METHOD lockstep_move_max
VAR_INPUT
	LockstepGroup	: USINT := 1; // The address of the lockstep group must be in the range 1 to lockstep.numgroups; lockstep.numgroups: the number of lockstep groupss; Valid Values: 0 to 2
	max_speed 		: UDINT := ZaberConfiguration.MaxDynamics.Velocity;
	accel			: UDINT	:= ZaberConfiguration.MaxDynamics.Accel;
END_VAR
IF ZaberStatus.ComponentStatus.iLastCommand <> 0 THEN
	ZaberStatus.ComponentStatus.iLastCommand.P_CommandStatus.LastCommandMessage := Base.F_GetLastWordInString(__POUNAME());
END_IF

IF NOT _DispatchValid() THEN
	RETURN;
ELSE
	_ClearTempString();
	ZaberCommand.stringval := Tc2_Standard.CONCAT(STR1 := ZaberConfiguration.sControllerRef, STR2 := ' ');
	ZaberCommand.stringval := Tc2_Standard.CONCAT(STR1 := ZaberCommand.stringval, STR2 := Base.F_GetFirstWordInString(sInput := SUPER^._iCommandConfiguration[ZaberStatus.ZaberMethodDispatch].P_CommandConfiguration.CommandDescription));
	ZaberCommand.stringval := Tc2_Standard.CONCAT(STR1 := ZaberCommand.stringval, STR2 := ' ');
	ZaberCommand.stringval := Tc2_Standard.CONCAT(STR1 := ZaberCommand.stringval, STR2 := USINT_TO_STRING(LockstepGroup));
	ZaberCommand.stringval := Tc2_Standard.CONCAT(STR1 := ZaberCommand.stringval, STR2 := ' ');
	ZaberCommand.stringval := Tc2_Standard.CONCAT(STR1 := ZaberCommand.stringval, STR2 := F_GetAllButFirstWord(sInput := SUPER^._iCommandConfiguration[ZaberStatus.ZaberMethodDispatch].P_CommandConfiguration.CommandDescription));
	ZaberCommand.stringval := Tc2_Standard.CONCAT(STR1 := ZaberCommand.stringval, STR2 := ' ');
	ZaberCommand.stringval := Tc2_Standard.CONCAT(STR1 := ZaberCommand.stringval, STR2 := UDINT_TO_STRING(max_speed));
	ZaberCommand.stringval := Tc2_Standard.CONCAT(STR1 := ZaberCommand.stringval, STR2 := ' ');
	ZaberCommand.stringval := Tc2_Standard.CONCAT(STR1 := ZaberCommand.stringval, STR2 := UDINT_TO_STRING(accel));
	
	IF iBufferSend <> 0 AND __QUERYINTERFACE(iBufferSend, testIBufferSend) THEN
		iBufferSend.AddObject(RefObject := ZaberCommand);
	END_IF
END_IF
END_METHOD

METHOD lockstep_move_min
VAR_INPUT
	LockstepGroup	: USINT := 1; // The address of the lockstep group must be in the range 1 to lockstep.numgroups; lockstep.numgroups: the number of lockstep groupss; Valid Values: 0 to 2
	max_speed 		: UDINT := ZaberConfiguration.MaxDynamics.Velocity;
	accel			: UDINT := ZaberConfiguration.MaxDynamics.Accel;
END_VAR
IF ZaberStatus.ComponentStatus.iLastCommand <> 0 THEN
	ZaberStatus.ComponentStatus.iLastCommand.P_CommandStatus.LastCommandMessage := Base.F_GetLastWordInString(__POUNAME());
END_IF

IF NOT _DispatchValid() THEN
	RETURN;
ELSE
	_ClearTempString();
	ZaberCommand.stringval := Tc2_Standard.CONCAT(STR1 := ZaberConfiguration.sControllerRef, STR2 := ' ');
	ZaberCommand.stringval := Tc2_Standard.CONCAT(STR1 := ZaberCommand.stringval, STR2 := Base.F_GetFirstWordInString(sInput := SUPER^._iCommandConfiguration[ZaberStatus.ZaberMethodDispatch].P_CommandConfiguration.CommandDescription));
	ZaberCommand.stringval := Tc2_Standard.CONCAT(STR1 := ZaberCommand.stringval, STR2 := ' ');
	ZaberCommand.stringval := Tc2_Standard.CONCAT(STR1 := ZaberCommand.stringval, STR2 := USINT_TO_STRING(LockstepGroup));
	ZaberCommand.stringval := Tc2_Standard.CONCAT(STR1 := ZaberCommand.stringval, STR2 := ' ');
	ZaberCommand.stringval := Tc2_Standard.CONCAT(STR1 := ZaberCommand.stringval, STR2 := F_GetAllButFirstWord(sInput := SUPER^._iCommandConfiguration[ZaberStatus.ZaberMethodDispatch].P_CommandConfiguration.CommandDescription));
	ZaberCommand.stringval := Tc2_Standard.CONCAT(STR1 := ZaberCommand.stringval, STR2 := ' ');
	ZaberCommand.stringval := Tc2_Standard.CONCAT(STR1 := ZaberCommand.stringval, STR2 := UDINT_TO_STRING(max_speed));
	ZaberCommand.stringval := Tc2_Standard.CONCAT(STR1 := ZaberCommand.stringval, STR2 := ' ');
	ZaberCommand.stringval := Tc2_Standard.CONCAT(STR1 := ZaberCommand.stringval, STR2 := UDINT_TO_STRING(accel));
	
	IF iBufferSend <> 0 AND __QUERYINTERFACE(iBufferSend, testIBufferSend) THEN
		iBufferSend.AddObject(RefObject := ZaberCommand);
	END_IF
END_IF
END_METHOD

METHOD lockstep_move_sin
VAR_INPUT
	LockstepGroup	: USINT := 1; // The address of the lockstep group must be in the range 1 to lockstep.numgroups; lockstep.numgroups: the number of lockstep groupss; Valid Values: 0 to 2
	amplitude		: LREAL := ZaberConfiguration.SinParameters.Amplitude; // Amplitude of the sinusoidal motion
	period	 		: LREAL := ZaberConfiguration.SinParameters.Period; // Period of the sinusoidal motion in milliseconds and to one decimal place; Must be in the range 0.2 to 429,496,729.5
	count			: LREAL := ZaberConfiguration.SinParameters.Count; // Number of repeated cycles (optional); Must be a multiple of 0.5 in the range 0.5 to 2,147,483,647 (versions 7.29 and above)
END_VAR
IF ZaberStatus.ComponentStatus.iLastCommand <> 0 THEN
	ZaberStatus.ComponentStatus.iLastCommand.P_CommandStatus.LastCommandMessage := Base.F_GetLastWordInString(__POUNAME());
END_IF

IF NOT _DispatchValid() THEN
	RETURN;
ELSE
	_ClearTempString();
	ZaberCommand.stringval := Tc2_Standard.CONCAT(STR1 := ZaberConfiguration.sControllerRef, STR2 := ' ');
	ZaberCommand.stringval := Tc2_Standard.CONCAT(STR1 := ZaberCommand.stringval, STR2 := Base.F_GetFirstWordInString(sInput := SUPER^._iCommandConfiguration[ZaberStatus.ZaberMethodDispatch].P_CommandConfiguration.CommandDescription));
	ZaberCommand.stringval := Tc2_Standard.CONCAT(STR1 := ZaberCommand.stringval, STR2 := ' ');
	ZaberCommand.stringval := Tc2_Standard.CONCAT(STR1 := ZaberCommand.stringval, STR2 := USINT_TO_STRING(LockstepGroup));
	ZaberCommand.stringval := Tc2_Standard.CONCAT(STR1 := ZaberCommand.stringval, STR2 := ' ');
	ZaberCommand.stringval := Tc2_Standard.CONCAT(STR1 := ZaberCommand.stringval, STR2 := F_GetAllButFirstWord(sInput := SUPER^._iCommandConfiguration[ZaberStatus.ZaberMethodDispatch].P_CommandConfiguration.CommandDescription));
	ZaberCommand.stringval := Tc2_Standard.CONCAT(STR1 := ZaberCommand.stringval, STR2 := ' ');
	ZaberCommand.stringval := Tc2_Standard.CONCAT(STR1 := ZaberCommand.stringval, STR2 := LREAL_TO_STRING(amplitude));
	ZaberCommand.stringval := Tc2_Standard.CONCAT(STR1 := ZaberCommand.stringval, STR2 := ' ');
	ZaberCommand.stringval := Tc2_Standard.CONCAT(STR1 := ZaberCommand.stringval, STR2 := LREAL_TO_STRING(period));
	ZaberCommand.stringval := Tc2_Standard.CONCAT(STR1 := ZaberCommand.stringval, STR2 := ' ');
	ZaberCommand.stringval := Tc2_Standard.CONCAT(STR1 := ZaberCommand.stringval, STR2 := LREAL_TO_STRING(count));
	
	IF iBufferSend <> 0 AND __QUERYINTERFACE(iBufferSend, testIBufferSend) THEN
		iBufferSend.AddObject(RefObject := ZaberCommand);
	END_IF
END_IF
END_METHOD

METHOD move_abs
VAR_INPUT
	position	: UDINT := ZaberConfiguration.SetDynamics.Position;
	max_speed 	: UDINT := ZaberConfiguration.MaxDynamics.Velocity;
	accel		: UDINT := ZaberConfiguration.MaxDynamics.Accel;
END_VAR
IF ZaberStatus.ComponentStatus.iLastCommand <> 0 THEN
	ZaberStatus.ComponentStatus.iLastCommand.P_CommandStatus.LastCommandMessage := Base.F_GetLastWordInString(__POUNAME());
END_IF

IF NOT _DispatchValid() THEN
	RETURN;
ELSE
	_BuildCommandStringNoArgs();
	ZaberCommand.stringval := Tc2_Standard.CONCAT(STR1 := ZaberCommand.stringval, STR2 := ' ');
	ZaberCommand.stringval := Tc2_Standard.CONCAT(STR1 := ZaberCommand.stringval, STR2 := UDINT_TO_STRING(position));
	ZaberCommand.stringval := Tc2_Standard.CONCAT(STR1 := ZaberCommand.stringval, STR2 := ' ');
	ZaberCommand.stringval := Tc2_Standard.CONCAT(STR1 := ZaberCommand.stringval, STR2 := UDINT_TO_STRING(max_speed));
	ZaberCommand.stringval := Tc2_Standard.CONCAT(STR1 := ZaberCommand.stringval, STR2 := ' ');
	ZaberCommand.stringval := Tc2_Standard.CONCAT(STR1 := ZaberCommand.stringval, STR2 := UDINT_TO_STRING(accel));

	IF iBufferSend <> 0 AND __QUERYINTERFACE(iBufferSend, testIBufferSend) THEN
		iBufferSend.AddObject(RefObject := ZaberCommand);
	END_IF
END_IF
END_METHOD

METHOD move_index_next
IF ZaberStatus.ComponentStatus.iLastCommand <> 0 THEN
	ZaberStatus.ComponentStatus.iLastCommand.P_CommandStatus.LastCommandMessage := Base.F_GetLastWordInString(__POUNAME());
END_IF

IF NOT _DispatchValid() THEN
	RETURN;
ELSE
	_BuildCommandStringNoArgs();
	
	IF iBufferSend <> 0 AND __QUERYINTERFACE(iBufferSend, testIBufferSend) THEN
		iBufferSend.AddObject(RefObject := ZaberCommand);
	END_IF
END_IF
END_METHOD

METHOD move_index_prev
IF ZaberStatus.ComponentStatus.iLastCommand <> 0 THEN
	ZaberStatus.ComponentStatus.iLastCommand.P_CommandStatus.LastCommandMessage := Base.F_GetLastWordInString(__POUNAME());
END_IF

IF NOT _DispatchValid() THEN
	RETURN;
ELSE
	_BuildCommandStringNoArgs();
	
	IF iBufferSend <> 0 AND __QUERYINTERFACE(iBufferSend, testIBufferSend) THEN
		iBufferSend.AddObject(RefObject := ZaberCommand);
	END_IF
END_IF
END_METHOD

METHOD move_max
IF ZaberStatus.ComponentStatus.iLastCommand <> 0 THEN
	ZaberStatus.ComponentStatus.iLastCommand.P_CommandStatus.LastCommandMessage := Base.F_GetLastWordInString(__POUNAME());
END_IF

IF NOT _DispatchValid() THEN
	RETURN;
ELSE
	_BuildCommandStringNoArgs();
	
	IF iBufferSend <> 0 AND __QUERYINTERFACE(iBufferSend, testIBufferSend) THEN
		iBufferSend.AddObject(RefObject := ZaberCommand);
	END_IF
END_IF
END_METHOD

METHOD move_min
IF ZaberStatus.ComponentStatus.iLastCommand <> 0 THEN
	ZaberStatus.ComponentStatus.iLastCommand.P_CommandStatus.LastCommandMessage := Base.F_GetLastWordInString(__POUNAME());
END_IF

IF NOT _DispatchValid() THEN
	RETURN;
ELSE
	_BuildCommandStringNoArgs();
	
	IF iBufferSend <> 0 AND __QUERYINTERFACE(iBufferSend, testIBufferSend) THEN
		iBufferSend.AddObject(RefObject := ZaberCommand);
	END_IF
END_IF
END_METHOD

METHOD move_scan_track_once
IF ZaberStatus.ComponentStatus.iLastCommand <> 0 THEN
	ZaberStatus.ComponentStatus.iLastCommand.P_CommandStatus.LastCommandMessage := Base.F_GetLastWordInString(__POUNAME());
END_IF

IF NOT _DispatchValid() THEN
	RETURN;
ELSE
	_BuildCommandStringNoArgs();
	
	IF iBufferSend <> 0 AND __QUERYINTERFACE(iBufferSend, testIBufferSend) THEN
		iBufferSend.AddObject(RefObject := ZaberCommand);
	END_IF
END_IF
END_METHOD

METHOD move_sin
VAR_INPUT
	amplitude		: LREAL; // Amplitude of the sinusoidal motion
	period	 		: LREAL; // Period of the sinusoidal motion in milliseconds and to one decimal place; Must be in the range 0.2 to 429,496,729.5
	count			: LREAL; // Number of repeated cycles (optional); Must be a multiple of 0.5 in the range 0.5 to 2,147,483,647 (versions 7.29 and above)
END_VAR
IF ZaberStatus.ComponentStatus.iLastCommand <> 0 THEN
	ZaberStatus.ComponentStatus.iLastCommand.P_CommandStatus.LastCommandMessage := Base.F_GetLastWordInString(__POUNAME());
END_IF

IF NOT _DispatchValid() THEN
	RETURN;
ELSE
	_ClearTempString();
	ZaberCommand.stringval := Tc2_Standard.CONCAT(STR1 := ZaberConfiguration.sControllerRef, STR2 := ' ');
	ZaberCommand.stringval := Tc2_Standard.CONCAT(STR1 := ZaberCommand.stringval, STR2 := UINT_TO_STRING(ZaberConfiguration.AxisRef));
	ZaberCommand.stringval := Tc2_Standard.CONCAT(STR1 := ZaberCommand.stringval, STR2 := ' ');
	ZaberCommand.stringval := Tc2_Standard.CONCAT(STR1 := ZaberCommand.stringval, STR2 := SUPER^._iCommandConfiguration[ZaberStatus.ZaberMethodDispatch].P_CommandConfiguration.CommandDescription);
	ZaberCommand.stringval := Tc2_Standard.CONCAT(STR1 := ZaberCommand.stringval, STR2 := ' ');
	ZaberCommand.stringval := Tc2_Standard.CONCAT(STR1 := ZaberCommand.stringval, STR2 := LREAL_TO_STRING(amplitude));
	ZaberCommand.stringval := Tc2_Standard.CONCAT(STR1 := ZaberCommand.stringval, STR2 := ' ');
	ZaberCommand.stringval := Tc2_Standard.CONCAT(STR1 := ZaberCommand.stringval, STR2 := LREAL_TO_STRING(period));
	ZaberCommand.stringval := Tc2_Standard.CONCAT(STR1 := ZaberCommand.stringval, STR2 := ' ');
	ZaberCommand.stringval := Tc2_Standard.CONCAT(STR1 := ZaberCommand.stringval, STR2 := LREAL_TO_STRING(count));
	
	IF iBufferSend <> 0 AND __QUERYINTERFACE(iBufferSend, testIBufferSend) THEN
		iBufferSend.AddObject(RefObject := ZaberCommand);
	END_IF
END_IF
END_METHOD

METHOD move_track
IF ZaberStatus.ComponentStatus.iLastCommand <> 0 THEN
	ZaberStatus.ComponentStatus.iLastCommand.P_CommandStatus.LastCommandMessage := Base.F_GetLastWordInString(__POUNAME());
END_IF

IF NOT _DispatchValid() THEN
	RETURN;
ELSE
	_BuildCommandStringNoArgs();
	
	IF iBufferSend <> 0 AND __QUERYINTERFACE(iBufferSend, testIBufferSend) THEN
		iBufferSend.AddObject(RefObject := ZaberCommand);
	END_IF
END_IF
END_METHOD

METHOD move_vel
VAR_INPUT
	velocity		: DINT;
	accel			: UDINT;
END_VAR
IF ZaberStatus.ComponentStatus.iLastCommand <> 0 THEN
	ZaberStatus.ComponentStatus.iLastCommand.P_CommandStatus.LastCommandMessage := Base.F_GetLastWordInString(__POUNAME());
END_IF

IF NOT _DispatchValid() THEN
	RETURN;
ELSE
	_ClearTempString();
	ZaberCommand.stringval := Tc2_Standard.CONCAT(STR1 := ZaberConfiguration.sControllerRef, STR2 := ' ');
	ZaberCommand.stringval := Tc2_Standard.CONCAT(STR1 := ZaberCommand.stringval, STR2 := UINT_TO_STRING(ZaberConfiguration.AxisRef));
	ZaberCommand.stringval := Tc2_Standard.CONCAT(STR1 := ZaberCommand.stringval, STR2 := ' ');
	ZaberCommand.stringval := Tc2_Standard.CONCAT(STR1 := ZaberCommand.stringval, STR2 := SUPER^._iCommandConfiguration[ZaberStatus.ZaberMethodDispatch].P_CommandConfiguration.CommandDescription);
	ZaberCommand.stringval := Tc2_Standard.CONCAT(STR1 := ZaberCommand.stringval, STR2 := ' ');
	ZaberCommand.stringval := Tc2_Standard.CONCAT(STR1 := ZaberCommand.stringval, STR2 := DINT_TO_STRING(velocity));
	ZaberCommand.stringval := Tc2_Standard.CONCAT(STR1 := ZaberCommand.stringval, STR2 := ' ');
	ZaberCommand.stringval := Tc2_Standard.CONCAT(STR1 := ZaberCommand.stringval, STR2 := UDINT_TO_STRING(accel));
	
	IF iBufferSend <> 0 AND __QUERYINTERFACE(iBufferSend, testIBufferSend) THEN
		iBufferSend.AddObject(RefObject := ZaberCommand);
	END_IF
END_IF
END_METHOD

METHOD pvt_buffer_list
IF ZaberStatus.ComponentStatus.iLastCommand <> 0 THEN
	ZaberStatus.ComponentStatus.iLastCommand.P_CommandStatus.LastCommandMessage := Base.F_GetLastWordInString(__POUNAME());
END_IF

IF NOT _DispatchValid() THEN
	RETURN;
ELSE
	_BuildCommandStringNoArgs();
	
	IF iBufferSend <> 0 AND __QUERYINTERFACE(iBufferSend, testIBufferSend) THEN
		iBufferSend.AddObject(RefObject := ZaberCommand);
	END_IF
END_IF
END_METHOD

METHOD renumber
IF ZaberStatus.ComponentStatus.iLastCommand <> 0 THEN
	ZaberStatus.ComponentStatus.iLastCommand.P_CommandStatus.LastCommandMessage := Base.F_GetLastWordInString(__POUNAME());
END_IF

IF NOT _DispatchValid() THEN
	RETURN;
ELSE
	_BuildCommandStringNoArgs();
	
	IF iBufferSend <> 0 AND __QUERYINTERFACE(iBufferSend, testIBufferSend) THEN
		iBufferSend.AddObject(RefObject := ZaberCommand);
	END_IF
END_IF
END_METHOD

METHOD scope_clear
IF ZaberStatus.ComponentStatus.iLastCommand <> 0 THEN
	ZaberStatus.ComponentStatus.iLastCommand.P_CommandStatus.LastCommandMessage := Base.F_GetLastWordInString(__POUNAME());
END_IF

IF NOT _DispatchValid() THEN
	RETURN;
ELSE
	_BuildCommandStringNoArgs();
	
	IF iBufferSend <> 0 AND __QUERYINTERFACE(iBufferSend, testIBufferSend) THEN
		iBufferSend.AddObject(RefObject := ZaberCommand);
	END_IF
END_IF
END_METHOD

METHOD scope_print
IF ZaberStatus.ComponentStatus.iLastCommand <> 0 THEN
	ZaberStatus.ComponentStatus.iLastCommand.P_CommandStatus.LastCommandMessage := Base.F_GetLastWordInString(__POUNAME());
END_IF

IF NOT _DispatchValid() THEN
	RETURN;
ELSE
	_BuildCommandStringNoArgs();
	
	IF iBufferSend <> 0 AND __QUERYINTERFACE(iBufferSend, testIBufferSend) THEN
		iBufferSend.AddObject(RefObject := ZaberCommand);
	END_IF
END_IF
END_METHOD

METHOD scope_stop
IF ZaberStatus.ComponentStatus.iLastCommand <> 0 THEN
	ZaberStatus.ComponentStatus.iLastCommand.P_CommandStatus.LastCommandMessage := Base.F_GetLastWordInString(__POUNAME());
END_IF

IF NOT _DispatchValid() THEN
	RETURN;
ELSE
	_BuildCommandStringNoArgs();
	
	IF iBufferSend <> 0 AND __QUERYINTERFACE(iBufferSend, testIBufferSend) THEN
		iBufferSend.AddObject(RefObject := ZaberCommand);
	END_IF
END_IF
END_METHOD

METHOD set_comm_checksum
VAR_INPUT
	Value	: INT := 1; //0 = Disabled, 1 = Enabled, 2 = Automatic
END_VAR
IF ZaberStatus.ComponentStatus.iLastCommand <> 0 THEN
	ZaberStatus.ComponentStatus.iLastCommand.P_CommandStatus.LastCommandMessage := Base.F_GetLastWordInString(__POUNAME());
END_IF

IF NOT _DispatchValid() THEN
	RETURN;
ELSE
	_BuildCommandStringNoArgs();
	ZaberCommand.stringval := Tc2_Standard.CONCAT(STR1 := ZaberCommand.stringval, STR2 := ' ');
	ZaberCommand.stringval := Tc2_Standard.CONCAT(STR1 := ZaberCommand.stringval, STR2 := INT_TO_STRING(Value));
	
	IF iBufferSend <> 0 AND __QUERYINTERFACE(iBufferSend, testIBufferSend) THEN
		iBufferSend.AddObject(RefObject := ZaberCommand);
	END_IF
END_IF
END_METHOD

METHOD stop
IF ZaberStatus.ComponentStatus.iLastCommand <> 0 THEN
	ZaberStatus.ComponentStatus.iLastCommand.P_CommandStatus.LastCommandMessage := Base.F_GetLastWordInString(__POUNAME());
END_IF

IF NOT _DispatchValid() THEN
	RETURN;
ELSE
	_BuildCommandStringNoArgs();
	
	IF iBufferSend <> 0 AND __QUERYINTERFACE(iBufferSend, testIBufferSend) THEN
		iBufferSend.AddObject(RefObject := ZaberCommand);
	END_IF
END_IF
END_METHOD

METHOD storage_erase
IF ZaberStatus.ComponentStatus.iLastCommand <> 0 THEN
	ZaberStatus.ComponentStatus.iLastCommand.P_CommandStatus.LastCommandMessage := Base.F_GetLastWordInString(__POUNAME());
END_IF

IF NOT _DispatchValid() THEN
	RETURN;
ELSE
	_BuildCommandStringNoArgs();
	
	IF iBufferSend <> 0 AND __QUERYINTERFACE(iBufferSend, testIBufferSend) THEN
		iBufferSend.AddObject(RefObject := ZaberCommand);
	END_IF
END_IF
END_METHOD

METHOD storage_print
IF ZaberStatus.ComponentStatus.iLastCommand <> 0 THEN
	ZaberStatus.ComponentStatus.iLastCommand.P_CommandStatus.LastCommandMessage := Base.F_GetLastWordInString(__POUNAME());
END_IF

IF NOT _DispatchValid() THEN
	RETURN;
ELSE
	_BuildCommandStringNoArgs();
	
	IF iBufferSend <> 0 AND __QUERYINTERFACE(iBufferSend, testIBufferSend) THEN
		iBufferSend.AddObject(RefObject := ZaberCommand);
	END_IF
END_IF
END_METHOD

METHOD stream_buffer_list
IF ZaberStatus.ComponentStatus.iLastCommand <> 0 THEN
	ZaberStatus.ComponentStatus.iLastCommand.P_CommandStatus.LastCommandMessage := Base.F_GetLastWordInString(__POUNAME());
END_IF

IF NOT _DispatchValid() THEN
	RETURN;
ELSE
	_BuildCommandStringNoArgs();
	
	IF iBufferSend <> 0 AND __QUERYINTERFACE(iBufferSend, testIBufferSend) THEN
		iBufferSend.AddObject(RefObject := ZaberCommand);
	END_IF
END_IF
END_METHOD

METHOD system_errors
IF ZaberStatus.ComponentStatus.iLastCommand <> 0 THEN
	ZaberStatus.ComponentStatus.iLastCommand.P_CommandStatus.LastCommandMessage := Base.F_GetLastWordInString(__POUNAME());
END_IF

IF NOT _DispatchValid() THEN
	RETURN;
ELSE
	_BuildCommandStringNoArgs();
	
	IF iBufferSend <> 0 AND __QUERYINTERFACE(iBufferSend, testIBufferSend) THEN
		iBufferSend.AddObject(RefObject := ZaberCommand);
	END_IF
END_IF
END_METHOD

METHOD system_factoryreset
IF ZaberStatus.ComponentStatus.iLastCommand <> 0 THEN
	ZaberStatus.ComponentStatus.iLastCommand.P_CommandStatus.LastCommandMessage := Base.F_GetLastWordInString(__POUNAME());
END_IF

IF NOT _DispatchValid() THEN
	RETURN;
ELSE
	_BuildCommandStringNoArgs();
	
	IF iBufferSend <> 0 AND __QUERYINTERFACE(iBufferSend, testIBufferSend) THEN
		iBufferSend.AddObject(RefObject := ZaberCommand);
	END_IF
END_IF
END_METHOD

METHOD system_reset
IF ZaberStatus.ComponentStatus.iLastCommand <> 0 THEN
	ZaberStatus.ComponentStatus.iLastCommand.P_CommandStatus.LastCommandMessage := Base.F_GetLastWordInString(__POUNAME());
END_IF

IF NOT _DispatchValid() THEN
	RETURN;
ELSE
	_BuildCommandStringNoArgs();
	
	IF iBufferSend <> 0 AND __QUERYINTERFACE(iBufferSend, testIBufferSend) THEN
		iBufferSend.AddObject(RefObject := ZaberCommand);
	END_IF
END_IF
END_METHOD

METHOD system_restore
IF ZaberStatus.ComponentStatus.iLastCommand <> 0 THEN
	ZaberStatus.ComponentStatus.iLastCommand.P_CommandStatus.LastCommandMessage := Base.F_GetLastWordInString(__POUNAME());
END_IF

IF NOT _DispatchValid() THEN
	RETURN;
ELSE
	_BuildCommandStringNoArgs();
	
	IF iBufferSend <> 0 AND __QUERYINTERFACE(iBufferSend, testIBufferSend) THEN
		iBufferSend.AddObject(RefObject := ZaberCommand);
	END_IF
END_IF
END_METHOD

METHOD tools_echo
IF ZaberStatus.ComponentStatus.iLastCommand <> 0 THEN
	ZaberStatus.ComponentStatus.iLastCommand.P_CommandStatus.LastCommandMessage := Base.F_GetLastWordInString(__POUNAME());
END_IF

IF NOT _DispatchValid() THEN
	RETURN;
ELSE
	_BuildCommandStringNoArgs();
	
	IF iBufferSend <> 0 AND __QUERYINTERFACE(iBufferSend, testIBufferSend) THEN
		iBufferSend.AddObject(RefObject := ZaberCommand);
	END_IF
END_IF
END_METHOD

METHOD tools_findrange
IF ZaberStatus.ComponentStatus.iLastCommand <> 0 THEN
	ZaberStatus.ComponentStatus.iLastCommand.P_CommandStatus.LastCommandMessage := Base.F_GetLastWordInString(__POUNAME());
END_IF

IF NOT _DispatchValid() THEN
	RETURN;
ELSE
	_BuildCommandStringNoArgs();
	
	IF iBufferSend <> 0 AND __QUERYINTERFACE(iBufferSend, testIBufferSend) THEN
		iBufferSend.AddObject(RefObject := ZaberCommand);
	END_IF
END_IF
END_METHOD

METHOD tools_gotolimit
IF ZaberStatus.ComponentStatus.iLastCommand <> 0 THEN
	ZaberStatus.ComponentStatus.iLastCommand.P_CommandStatus.LastCommandMessage := Base.F_GetLastWordInString(__POUNAME());
END_IF

IF NOT _DispatchValid() THEN
	RETURN;
ELSE
	_BuildCommandStringNoArgs();
	
	IF iBufferSend <> 0 AND __QUERYINTERFACE(iBufferSend, testIBufferSend) THEN
		iBufferSend.AddObject(RefObject := ZaberCommand);
	END_IF
END_IF
END_METHOD

METHOD tools_parking
IF ZaberStatus.ComponentStatus.iLastCommand <> 0 THEN
	ZaberStatus.ComponentStatus.iLastCommand.P_CommandStatus.LastCommandMessage := Base.F_GetLastWordInString(__POUNAME());
END_IF

IF NOT _DispatchValid() THEN
	RETURN;
ELSE
	_BuildCommandStringNoArgs();
	
	IF iBufferSend <> 0 AND __QUERYINTERFACE(iBufferSend, testIBufferSend) THEN
		iBufferSend.AddObject(RefObject := ZaberCommand);
	END_IF
END_IF
END_METHOD

METHOD tools_setcomm
IF ZaberStatus.ComponentStatus.iLastCommand <> 0 THEN
	ZaberStatus.ComponentStatus.iLastCommand.P_CommandStatus.LastCommandMessage := Base.F_GetLastWordInString(__POUNAME());
END_IF

IF NOT _DispatchValid() THEN
	RETURN;
ELSE
	_BuildCommandStringNoArgs();
	
	IF iBufferSend <> 0 AND __QUERYINTERFACE(iBufferSend, testIBufferSend) THEN
		iBufferSend.AddObject(RefObject := ZaberCommand);
	END_IF
END_IF
END_METHOD

METHOD tools_storepos_current
IF ZaberStatus.ComponentStatus.iLastCommand <> 0 THEN
	ZaberStatus.ComponentStatus.iLastCommand.P_CommandStatus.LastCommandMessage := Base.F_GetLastWordInString(__POUNAME());
END_IF

IF NOT _DispatchValid() THEN
	RETURN;
ELSE
	_BuildCommandStringNoArgs();
	
	IF iBufferSend <> 0 AND __QUERYINTERFACE(iBufferSend, testIBufferSend) THEN
		iBufferSend.AddObject(RefObject := ZaberCommand);
	END_IF
END_IF
END_METHOD

METHOD tools_storepos_position
IF ZaberStatus.ComponentStatus.iLastCommand <> 0 THEN
	ZaberStatus.ComponentStatus.iLastCommand.P_CommandStatus.LastCommandMessage := Base.F_GetLastWordInString(__POUNAME());
END_IF

IF NOT _DispatchValid() THEN
	RETURN;
ELSE
	_BuildCommandStringNoArgs();
	
	IF iBufferSend <> 0 AND __QUERYINTERFACE(iBufferSend, testIBufferSend) THEN
		iBufferSend.AddObject(RefObject := ZaberCommand);
	END_IF
END_IF
END_METHOD

METHOD trigger_print
IF ZaberStatus.ComponentStatus.iLastCommand <> 0 THEN
	ZaberStatus.ComponentStatus.iLastCommand.P_CommandStatus.LastCommandMessage := Base.F_GetLastWordInString(__POUNAME());
END_IF

IF NOT _DispatchValid() THEN
	RETURN;
ELSE
	_BuildCommandStringNoArgs();
	
	IF iBufferSend <> 0 AND __QUERYINTERFACE(iBufferSend, testIBufferSend) THEN
		iBufferSend.AddObject(RefObject := ZaberCommand);
	END_IF
END_IF
END_METHOD

METHOD trigger_show
IF ZaberStatus.ComponentStatus.iLastCommand <> 0 THEN
	ZaberStatus.ComponentStatus.iLastCommand.P_CommandStatus.LastCommandMessage := Base.F_GetLastWordInString(__POUNAME());
END_IF

IF NOT _DispatchValid() THEN
	RETURN;
ELSE
	_BuildCommandStringNoArgs();
	
	IF iBufferSend <> 0 AND __QUERYINTERFACE(iBufferSend, testIBufferSend) THEN
		iBufferSend.AddObject(RefObject := ZaberCommand);
	END_IF
END_IF
END_METHOD

METHOD trigger_when_dist
IF ZaberStatus.ComponentStatus.iLastCommand <> 0 THEN
	ZaberStatus.ComponentStatus.iLastCommand.P_CommandStatus.LastCommandMessage := Base.F_GetLastWordInString(__POUNAME());
END_IF

IF NOT _DispatchValid() THEN
	RETURN;
ELSE
	_BuildCommandStringNoArgs();
	
	IF iBufferSend <> 0 AND __QUERYINTERFACE(iBufferSend, testIBufferSend) THEN
		iBufferSend.AddObject(RefObject := ZaberCommand);
	END_IF
END_IF
END_METHOD

METHOD trigger_when_encoder_dist
IF ZaberStatus.ComponentStatus.iLastCommand <> 0 THEN
	ZaberStatus.ComponentStatus.iLastCommand.P_CommandStatus.LastCommandMessage := Base.F_GetLastWordInString(__POUNAME());
END_IF

IF NOT _DispatchValid() THEN
	RETURN;
ELSE
	_BuildCommandStringNoArgs();
	
	IF iBufferSend <> 0 AND __QUERYINTERFACE(iBufferSend, testIBufferSend) THEN
		iBufferSend.AddObject(RefObject := ZaberCommand);
	END_IF
END_IF
END_METHOD

METHOD warnings
IF ZaberStatus.ComponentStatus.iLastCommand <> 0 THEN
	ZaberStatus.ComponentStatus.iLastCommand.P_CommandStatus.LastCommandMessage := Base.F_GetLastWordInString(__POUNAME());
END_IF

IF NOT _DispatchValid() THEN
	RETURN;
ELSE
	_BuildCommandStringNoArgs();
	
	IF iBufferSend <> 0 AND __QUERYINTERFACE(iBufferSend, testIBufferSend) THEN
		iBufferSend.AddObject(RefObject := ZaberCommand);
	END_IF
END_IF
END_METHOD

METHOD warnings_clear
IF ZaberStatus.ComponentStatus.iLastCommand <> 0 THEN
	ZaberStatus.ComponentStatus.iLastCommand.P_CommandStatus.LastCommandMessage := Base.F_GetLastWordInString(__POUNAME());
END_IF

IF NOT _DispatchValid() THEN
	RETURN;
ELSE
	_BuildCommandStringNoArgs();
	
	IF iBufferSend <> 0 AND __QUERYINTERFACE(iBufferSend, testIBufferSend) THEN
		iBufferSend.AddObject(RefObject := ZaberCommand);
	END_IF
END_IF
END_METHOD

METHOD CyclicLogic
SUPER^.CyclicLogic();

_ConfigurationCyclic();

_DebugTesting();

ftRun(CLK := Run);
IF ftRun.Q THEN
	stop();
END_IF

_SendCyclic();

_ReceiveCyclic();

IF ZaberConfiguration.EnablePollingOnMotion THEN
	IF (ZaberStatus.ZaberReply.MotionStatus = 'BUSY') THEN
		_PollBusy();
	END_IF
END_IF
END_METHOD

{attribute 'monitoring' := 'call'}
PROPERTY P_ZaberConfiguration : REFERENCE TO ST_ZaberConfiguration
GET
P_ZaberConfiguration REF= _ResolveZaberConfiguration();
END_GET
END_PROPERTY

(* Basic component initialization logic*)
METHOD PROTECTED _Initialize : BOOL
SUPER^.BaseStatus.Initialized := _InitializeChildrenDependencies();

SUPER^.BaseStatus.Initialized	:= _InitializeReferences();

SUPER^.BaseStatus.Busy	:= FALSE;

_SetCommandIndices();

_ResolveZaberConfiguration();

// IF _InterfacesInjectable() THEN
// 	_InjectDependencies();
// END_IF

IF SUPER^.ComponentConfiguration.AmsNetIdRequired AND_THEN NOT SUPER^.ComponentStatus.AmsNetIdIsValid THEN
	REPEAT
		_ObtainAmsNetId();
	UNTIL SUPER^.ComponentStatus.AmsNetIdIsValid OR SUPER^.GetAmsNetId.bError
	END_REPEAT;

	IF SUPER^.GetAmsNetId.bError THEN
		IF SUPER^.BaseConfiguration.LogTraceConfiguration.What.xLogToEventLogger THEN
			TraceWithSeverity(Message := 'Error: Component failed to obtain AmsNetId', Severity := TcEventSeverity.Error);
		END_IF
	END_IF
END_IF

// Set InitSuccess only if requirement is satisfied or not required
IF (SUPER^.ComponentConfiguration.AmsNetIdRequired AND SUPER^.ComponentStatus.AmsNetIdIsValid)
   OR (NOT SUPER^.ComponentConfiguration.AmsNetIdRequired) THEN
	SUPER^.BaseStatus.Initialized := TRUE;
END_IF

IF NOT SUPER^.BaseStatus.Initialized AND SUPER^.BaseConfiguration.LogTraceConfiguration.What.xLogToEventLogger THEN
	TraceWithSeverity(Message := 'Initialization Failed - look at _Initialize method', Severity := TcEventSeverity.Error);
END_IF

IF SUPER^.BaseStatus.Initialized THEN
	_GetConfigParametersOnInit();
END_IF

_Initialize 	:= TRUE;
END_METHOD

METHOD PROTECTED _InitializeChildrenDependencies : BOOL
SUPER^._InitializeChildrenDependencies();

RingBufferSend.Initialize();
RingBufferRcv.Initialize();
RingBufferAll.Initialize();

_InitializeChildrenDependencies := TRUE;
END_METHOD

METHOD PROTECTED _InitializeReferences : BOOL
//Initialize data references
SUPER^._InitializeReferences();

SUPER^.ComponentConfiguration.BaseConfiguration 			REF= SUPER^.BaseConfiguration;
                                                    
SUPER^.ComponentStatus.BaseStatus							REF= SUPER^.BaseStatus;

ZaberConfiguration.ComponentConfiguration					REF= SUPER^.ComponentConfiguration;

ZaberStatus.ComponentStatus									REF= SUPER^.ComponentStatus;

_InitializeReferences 								:= TRUE; // apply at end of all reference initialization
END_METHOD

(*FB_Init is always available implicitly and it is used primarily for initialization.
The return value is not evaluated. For a specific influence, you can also declare the
methods explicitly and provide additional code there with the standard initialization
code. You can evaluate the return value.*)
METHOD FB_Init : BOOL
VAR_INPUT
	(* TRUE: the retain variables are initialized (reset warm / reset cold)*)
	bInitRetains	: BOOL;
	(* TRUE: the instance will be copied to the copy code afterward (online change)*)
	bInCopyCode	: BOOL;
END_VAR
END_METHOD

METHOD InjectDependencies : BOOL
VAR_INPUT
	SystemPermIntlk					: Base.I_PermIntlk;
	ControlMode						: Base.I_ControlMode;
	iSerialTx						: Communication.I_StringCmdStatusTx;
	iSerialRx						: Communication.I_StringCmdStatusRx;
	iSerialConfiguration			: Communication.I_SerialConfiguration;
	iSerialStatus					: Communication.I_SerialStatus;
END_VAR
//Serial Communication interfaces
_iSerialTx						:= iSerialTx;
_iSerialRx						:= iSerialRx;
_iSerialConfiguration			:= iSerialConfiguration;
_iSerialStatus					:= iSerialStatus;

// SystemPermIntlk := ; // SUPER^
// ControlMode		:= ;  // SUPER^
END_METHOD

METHOD PROTECTED _BuildCommandStringNoArgs
_ClearTempString();
ZaberCommand.stringval := Tc2_Standard.CONCAT(STR1 := ZaberConfiguration.sControllerRef, STR2 := ' ');
ZaberCommand.stringval := Tc2_Standard.CONCAT(STR1 := ZaberCommand.stringval, STR2 := UINT_TO_STRING(ZaberConfiguration.AxisRef));
ZaberCommand.stringval := Tc2_Standard.CONCAT(STR1 := ZaberCommand.stringval, STR2 := ' ');
ZaberCommand.stringval := Tc2_Standard.CONCAT(STR1 := ZaberCommand.stringval, STR2 := SUPER^._iCommandConfiguration[ZaberStatus.ZaberMethodDispatch].P_CommandConfiguration.CommandDescription);
END_METHOD

METHOD PROTECTED _ClearTempString
ZaberCommand.stringval := '';
END_METHOD

METHOD PROTECTED _ConfigurationCyclic
SUPER^._ConfigurationCyclic();

IF _iSerialConfiguration <> 0 THEN
	IF __ISVALIDREF(_iSerialConfiguration.P_SerialConfiguration) THEN
		_iSerialConfiguration.P_SerialConfiguration.ConfigurationLineControlADS.ComSerialConfiguration.ComPort 	:= ZaberConfiguration.ConfiguredComPort;
		IF __ISVALIDREF(_iSerialConfiguration.P_SerialConfiguration.StringConfigurationTx) THEN
			_iSerialConfiguration.P_SerialConfiguration.StringConfigurationTx.TxSuffix 							:= ZaberConfiguration.ConfiguredTerminationTx;
		END_IF
		IF __ISVALIDREF(_iSerialConfiguration.P_SerialConfiguration.StringConfigurationRx) THEN
			_iSerialConfiguration.P_SerialConfiguration.StringConfigurationRx.RxSuffix							:= ZaberConfiguration.ConfiguredTerminationRx;
		END_IF
		_iSerialConfiguration.P_SerialConfiguration.Enable														:= ZaberConfiguration.EnableSerialInterface;
	END_IF
END_IF

_ResolveZaberConfiguration();
END_METHOD

METHOD PRIVATE _DebugTesting
IF TrigCmd THEN
	IF _ZaberAxisConfigurationFW744 <> 0 THEN
		TempHash := _ZaberAxisConfigurationFW744.GetIndexByPOUName(NameIn := TempPouName);
	END_IF
	ExecuteCommand(CmdIndex := TempHash);
	TrigCmd := FALSE;
END_IF
END_METHOD

METHOD PROTECTED _DispatchValid : BOOL;
// Default to failure unless all checks pass
_DispatchValid := FALSE;

// Step 1: Out-of-bounds? Try rehash
IF NOT ((ZaberStatus.ZaberMethodDispatch >= LOWER_BOUND(SUPER^.Commands, 1)) AND
        (ZaberStatus.ZaberMethodDispatch <= UPPER_BOUND(SUPER^.Commands, 1))) THEN
    TraceWithSeverity('Dispatch index out of range � attempting re-hash', TcEventSeverity.Warning);

    IF ZaberStatus.ComponentStatus.iLastCommand <> 0 AND NOT _TryRehashDispatchIndex(ZaberStatus.ComponentStatus.iLastCommand.P_CommandStatus.LastCommandMessage) THEN
        RETURN;
    END_IF
END_IF

// Step 2: Mismatch? Try rehash again
IF ZaberStatus.ComponentStatus.iLastCommand <> 0 AND SUPER^._iCommandConfiguration[ZaberStatus.ZaberMethodDispatch]
        .P_CommandConfiguration.CommandPOUName <>
        ZaberStatus.ComponentStatus.iLastCommand.P_CommandStatus.LastCommandMessage THEN
    TraceWithSeverity('POU index mismatch � re-hashing', TcEventSeverity.Warning);

    IF ZaberStatus.ComponentStatus.iLastCommand <> 0 AND NOT _TryRehashDispatchIndex(ZaberStatus.ComponentStatus.iLastCommand.P_CommandStatus.LastCommandMessage) THEN
        RETURN;
    END_IF
END_IF

_DispatchValid := TRUE;
END_METHOD

METHOD PROTECTED _GetConfigParametersOnInit
//careful not to spam the serial interface with too much!
VAR

END_VAR
IF ZaberConfiguration.EnableGetParametersOnInit THEN
	// get_resolution();
	// WaitingForBits.WaitingForResolution	:= TRUE;
	//get_maxspeed();
	WaitingForBits.WaitingForMaxSpeed	:= TRUE;
END_IF
END_METHOD

METHOD PROTECTED _MapIndicesToCommands
CASE ZaberStatus.ZaberMethodDispatch OF

0:
    activate();
1:
    axis_restore();
2:
    driver_disable();
3:
    driver_enable();
4:
    home();
5:
    renumber();
6:
    stop();
7:
    warnings();
8:
    comm_en_ipv4_dhcp();
9:
    comm_en_ipv4_static();
10:
    io_cancel_schedule();
11:
    io_get_ai();
12:
    io_get_ao();
13:
    io_get_di();
14:
    io_get_do();
15:
    io_info();
16:
    io_set_ao();
17:
    io_set_ao_schedule();
18:
    io_set_do();
19:
    io_set_do_schedule();
20:
    move_abs(position := ZaberConfiguration.SetDynamics.Position, max_speed := ZaberConfiguration.MaxDynamics.Velocity, accel := ZaberConfiguration.MaxDynamics.Accel);
21:
    move_index();
22:
    move_index_next();
23:
    move_index_prev();
24:
    move_min();
25:
    move_max();
26:
    move_rel(max_speed := ZaberConfiguration.MaxDynamics.Velocity, distance := 100, accel := ZaberConfiguration.MaxDynamics.Accel);
27:
    move_scan_track_once();
28:
    move_sin(amplitude := ZaberConfiguration.SinParameters.Amplitude, period := ZaberConfiguration.SinParameters.Period, count := ZaberConfiguration.SinParameters.Count);
29:
    move_sin_stop();
30:
    move_stored();
31:
    move_track();
32:
    move_vel(velocity := ZaberConfiguration.SetDynamics.Velocity, accel := ZaberConfiguration.MaxDynamics.Accel);
33:
    lockstep_driver_disable(LockstepGroup := ZaberConfiguration.LockstepGroup);
34:
    lockstep_driver_enable(LockstepGroup := ZaberConfiguration.LockstepGroup);
35:
    lockstep_get(LockstepGroup := ZaberConfiguration.LockstepGroup, Setting := ZaberConfiguration.GetSetting);
36:
    lockstep_home(LockstepGroup := ZaberConfiguration.LockstepGroup);
37:
    lockstep_move_abs(LockstepGroup := ZaberConfiguration.LockstepGroup, max_speed := ZaberConfiguration.MaxDynamics.Velocity, position := ZaberConfiguration.SetDynamics.Position, accel := ZaberConfiguration.MaxDynamics.Accel);
38:
    lockstep_move_min(LockstepGroup := ZaberConfiguration.LockstepGroup, max_speed := ZaberConfiguration.MaxDynamics.Velocity, accel := ZaberConfiguration.MaxDynamics.Accel);
39:
    lockstep_move_max(LockstepGroup := ZaberConfiguration.LockstepGroup, max_speed := ZaberConfiguration.MaxDynamics.Velocity, accel := ZaberConfiguration.MaxDynamics.Accel);
40:
    lockstep_move_rel(LockstepGroup := ZaberConfiguration.LockstepGroup, distance := (ZaberConfiguration.SetDynamics.Position - ZaberStatus.Position), max_speed := ZaberConfiguration.MaxDynamics.Velocity, accel := ZaberConfiguration.MaxDynamics.Accel);
41:
    lockstep_move_sin(LockstepGroup := ZaberConfiguration.LockstepGroup, amplitude := ZaberConfiguration.SinParameters.Amplitude, period := ZaberConfiguration.SinParameters.Period, count := ZaberConfiguration.SinParameters.Count);
42:
    lockstep_move_sin_stop(LockstepGroup := ZaberConfiguration.LockstepGroup);
43:
    lockstep_move_stored();
44:
    lockstep_move_vel(LockstepGroup := ZaberConfiguration.LockstepGroup, accel := ZaberConfiguration.MaxDynamics.Accel, velocity := ZaberConfiguration.SetDynamics.Velocity);
45:
    lockstep_park(LockstepGroup := ZaberConfiguration.LockstepGroup);
46:
    lockstep_unpark(LockstepGroup := ZaberConfiguration.LockstepGroup);
47:
    lockstep_print(LockstepGroup := ZaberConfiguration.LockstepGroup);
48:
    lockstep_set_tolerance();
49:
    lockstep_setup_disable();
50:
    lockstep_setup_enable();
51:
    lockstep_stop(LockstepGroup := ZaberConfiguration.LockstepGroup);
52:
    pvt_buffer_erase();
53:
    pvt_buffer_list();
54:
    pvt_buffer_print();
55:
    pvt_call();
56:
    pvt_fifo();
57:
    pvt_info();
58:
    pvt_io_cancel_schedule();
59:
    pvt_io_set_ao();
60:
    pvt_io_set_ao_schedule();
61:
    pvt_io_set_do();
62:
    pvt_io_set_do_schedule();
63:
    pvt_point();
64:
    pvt_setup_disable();
65:
    pvt_setup_live();
66:
    pvt_setup_store();
67:
    scope_add();
68:
    scope_add_io_ai();
69:
    scope_add_io_ao();
70:
    scope_add_io_di();
71:
    scope_add_io_do();
72:
    scope_clear();
73:
    scope_print();
74:
    scope_start();
75:
    scope_stop();
76:
    storage_append();
77:
    storage_erase();
78:
    storage_exists();
79:
    storage_get();
80:
    storage_print();
81:
    storage_set();
82:
    stream_arc(StreamIndex := ZaberConfiguration.StreamNumber[0], Axis1 := ZaberConfiguration.ArcParameters.Axis1, Axis2 := ZaberConfiguration.ArcParameters.Axis2, 
				CenterX := ZaberConfiguration.ArcParameters.CenterX, CenterY := ZaberConfiguration.ArcParameters.CenterY, Direction := ZaberConfiguration.ArcParameters.Direction, EndX := ZaberConfiguration.ArcParameters.EndX, EndY := ZaberConfiguration.ArcParameters.EndY, 
				MoveType := ZaberConfiguration.ArcParameters.MoveType, Speed := ZaberConfiguration.SetDynamics.Velocity);
83:
    stream_buffer_erase();
84:
    stream_buffer_list();
85:
    stream_buffer_print();
86:
    stream_call();
87:
    stream_circle();
88:
    stream_fifo();
89:
    stream_helix();
90:
    stream_hold_onloff();
91:
    stream_info();
92:
    stream_io_cancel_schedule();
93:
    stream_io_set_ao();
94:
    stream_io_set_ao_schedule();
95:
    stream_io_set_do();
96:
    stream_io_set_do_schedule();
97:
    stream_line();
98:
    stream_set();
99:
    stream_setup_disable();
100:
    stream_setup_live(StreamNumber := 1, AxisNumber := ZaberConfiguration.AxisRef);
101:
    stream_setup_store(StreamNumber := ZaberConfiguration.StreamNumber[0], BufferNumber := ZaberConfiguration.BufferNumber, AxisNumber := ZaberConfiguration.AxisRef);
102:
    stream_wait();
103:
    stream_wait_io();
104:
    system_errors();
105:
    system_factoryreset();
106:
    system_reset();
107:
    system_restore();
108:
    tools_echo();
109:
    tools_findrange();
110:
    tools_gotolimit();
111:
    tools_parking();
112:
    tools_setcomm();
113:
    tools_storepos();
114:
    tools_storepos_current();
115:
    tools_storepos_position();
116:
    trigger_action_command();
117:
    trigger_action_none();
118:
    trigger_action_setting();
119:
    trigger_disable();
120:
    trigger_enable();
121:
    trigger_print();
122:
    trigger_show();
123:
    trigger_when_encoder_dist();
124:
    trigger_when_dist();
125:
    trigger_when_io();
126:
    trigger_when_setting();
127:
    trigger_when_time();
128:
    get_accel();
129:
    get_autodetect_coil_mode();
130:
    get_calibration_type();
131:
    get_comm_address();
132:
    get_comm_alert();
133:
    get_comm_checksum();
134:
    get_comm_command_packets_max();
135:
    get_comm_en_ipv4_address();
136:
    get_comm_en_ipv4_dhcp_enabled();
137:
    get_comm_en_ipv4_gateway();
138:
    get_comm_en_ipv4_netmask();
139:
    get_comm_en_mac();
140:
    get_comm_en_mdns_enable();
141:
    get_comm_next_owner();
142:
    get_comm_packet_size_max();
143:
    get_comm_protocol();
144:
    get_comm_rs232_baud();
145:
    get_comm_word_size_max();
146:
    get_device_hw_modified();
147:
    get_device_id();
148:
    get_driver_current_approach();
149:
    get_driver_current_hold();
150:
    get_driver_current_max();
151:
    get_driver_current_run();
152:
    get_driver_enable_mode();
153:
    get_driver_enabled();
154:
    get_driver_temperature();
155:
    get_get_settings_max();
156:
    get_ictrl_advance_a();
157:
    get_ictrl_advance_offset();
158:
    get_ictrl_afcff_inductance();
159:
    get_ictrl_afcff_ke();
160:
    get_ictrl_afcff_ki();
161:
    get_ictrl_afcff_max();
162:
    get_ictrl_afcff_ss();
163:
    get_ictrl_afcff_ss_max();
164:
    get_ictrl_delay();
165:
    get_ictrl_ff_kd();
166:
    get_ictrl_ff_kp();
167:
    get_ictrl_gain_coldmult();
168:
    get_ictrl_period();
169:
    get_ictrl_pi_ki();
170:
    get_ictrl_pi_kp();
171:
    get_ictrl_type();
172:
    get_io_ai_1_fc();
173:
    get_io_ai_2_fc();
174:
    get_io_ai_3_fc();
175:
    get_io_ai_4_fc();
176:
    get_io_di_port();
177:
    get_io_do_port();
178:
    get_knob_dir();
179:
    get_knob_distance();
180:
    get_knob_enable();
181:
    get_knob_maxspeed();
182:
    get_knob_mode();
183:
    get_knob_speedprofile();
184:
    get_limit_approach_maxspeed();
185:
    get_limit_detect_decelonly();
186:
    get_limit_detect_maxspeed();
187:
    get_limit_home_action();
188:
    get_limit_home_bidirectional();
189:
    get_limit_home_edge();
190:
    get_limit_home_offset();
191:
    get_limit_home_posupdate();
192:
    get_limit_home_preset();
193:
    get_limit_home_source();
194:
    get_limit_home_state();
195:
    get_limit_home_triggered();
196:
    get_limit_home_tune();
197:
    get_limit_home_type();
198:
    get_limit_home_width();
199:
    get_limit_max();
200:
    get_limit_min();
201:
    get_limit_range_mode();
202:
    get_lockstep_numgroups();
203:
    get_maxspeed();
204:
    get_motion_accel_ramptime();
205:
    get_motion_accelonly();
206:
    get_motion_busy();
207:
    get_motion_decelonly();
208:
    get_motion_index_dist();
209:
    get_motion_index_num();
210:
    get_motion_tracking_ai();
211:
    get_motion_tracking_dir();
212:
    get_motion_tracking_ki();
213:
    get_motion_tracking_kp();
214:
    get_motion_tracking_limit_max();
215:
    get_motion_tracking_limit_min();
216:
    get_motion_tracking_scan_dir();
217:
    get_motion_tracking_scan_maxspeed();
218:
    get_motion_tracking_scan_offset();
219:
    get_motion_tracking_scan_period();
220:
    get_motion_tracking_scan_signal_valid_delay();
221:
    get_motion_tracking_scan_tolerance();
222:
    get_motion_tracking_setpoint();
223:
    get_motion_tracking_settle_period();
224:
    get_motion_tracking_settle_tolerance();
225:
    get_motion_tracking_settle_tolerance_met();
226:
    get_motion_tracking_settled();
227:
    get_motion_tracking_signal_valid_di();
228:
    get_motor_current_max();
229:
    get_motor_inductance();
230:
    get_motor_ke();
231:
    get_motor_phase();
232:
    get_motor_phase_ratio_div1();
233:
    get_motor_phase_ratio_div2();
234:
    get_motor_phase_ratio_mult();
235:
    get_motor_resistance();
236:
    get_parking_state();
237:
    get_peripheral_hw_modified();
238:
    get_peripheral_id();
239:
    get_peripheral_id_pending();
240:
    get_peripheral_serial();
241:
    get_peripheral_serial_pending();
242:
    get_pos();
243:
    get_pvt_numseqs();
244:
    get_resolution();
245:
    get_scope_channel_size();
246:
    get_scope_channel_size_max();
247:
    get_scope_delay();
248:
    get_scope_numchannels();
249:
    get_scope_timebase();
250:
    get_stream_numbufs();
251:
    get_stream_numstreams();
252:
    get_system_access();
253:
    get_system_axiscount();
254:
    get_system_current_max();
255:
    get_system_led_enable();
256:
    get_system_serial();
257:
    get_system_temperature();
258:
    get_system_uptime();
259:
    get_system_voltage();
260:
    get_trigger_numactions();
261:
    get_trigger_numtriggers();
262:
    get_user_data_0();
263:
    get_user_data_1();
264:
    get_user_data_10();
265:
    get_user_data_11();
266:
    get_user_data_12();
267:
    get_user_data_13();
268:
    get_user_data_14();
269:
    get_user_data_15();
270:
    get_user_data_2();
271:
    get_user_data_3();
272:
    get_user_data_4();
273:
    get_user_data_5();
274:
    get_user_data_6();
275:
    get_user_data_7();
276:
    get_user_data_8();
277:
    get_user_data_9();
278:
    get_user_vdata_0();
279:
    get_user_vdata_1();
280:
    get_user_vdata_2();
281:
    get_user_vdata_3();
282:
    get_vel();
283:
    get_version();
284:
    get_version_build();
285:
    set_accel();
286:
    set_autodetect_coil_mode();
287:
    set_calibration_type();
288:
    set_comm_address();
289:
    set_comm_alert();
290:
    set_comm_checksum();
291:
    set_comm_command_packets_max();
292:
    set_comm_en_ipv4_address();
293:
    set_comm_en_ipv4_dhcp_enabled();
294:
    set_comm_en_ipv4_gateway();
295:
    set_comm_en_ipv4_netmask();
296:
    set_comm_en_mdns_enable();
297:
    set_comm_en_mac();
298:
    set_comm_next_owner();
299:
    set_comm_packet_size_max();
300:
    set_comm_protocol();
301:
    set_comm_rs232_baud();
302:
    set_comm_word_size_max();
303:
    set_driver_current_approach();
304:
    set_driver_current_hold();
305:
    set_driver_current_max();
306:
    set_driver_current_run();
307:
    set_driver_enable_mode();
308:
    set_driver_enabled();
309:
    set_driver_temperature();
310:
    set_get_settings_max();
311:
    set_ictrl_advance_a();
312:
    set_ictrl_advance_offset();
313:
    set_ictrl_afcff_inductance();
314:
    set_ictrl_afcff_ke();
315:
    set_ictrl_afcff_ki();
316:
    set_ictrl_afcff_max();
317:
    set_ictrl_afcff_ss();
318:
    set_ictrl_afcff_ss_max();
319:
    set_ictrl_delay();
320:
    set_ictrl_ff_kd();
321:
    set_ictrl_ff_kp();
322:
    set_ictrl_gain_coldmult();
323:
    set_ictrl_period();
324:
    set_ictrl_pi_ki();
325:
    set_ictrl_pi_kp();
326:
    set_ictrl_type();
327:
    set_io_ai_1_fc();
328:
    set_io_ai_2_fc();
329:
    set_io_ai_3_fc();
330:
    set_io_ai_4_fc();
331:
    set_io_di_port();
332:
    set_io_do_port();
333:
    set_knob_dir();
334:
    set_knob_distance();
335:
    set_knob_enable();
336:
    set_knob_maxspeed();
337:
    set_knob_mode();
338:
    set_knob_speedprofile();
339:
    set_limit_approach_maxspeed();
340:
    set_limit_detect_decelonly();
341:
    set_limit_detect_maxspeed();
342:
    set_limit_home_action();
343:
    set_limit_home_bidirectional();
344:
    set_limit_home_edge();
345:
    set_limit_home_offset();
346:
    set_limit_home_posupdate();
347:
    set_limit_home_preset();
348:
    set_limit_home_source();
349:
    set_limit_home_state();
350:
    set_limit_home_triggered();
351:
    set_limit_home_tune();
352:
    set_limit_home_type();
353:
    set_limit_home_width();
354:
    set_limit_max();
355:
    set_limit_min();
356:
    set_limit_range_mode();
357:
    set_lockstep_numgroups();
358:
    set_maxspeed();
359:
    set_motion_accel_ramptime();
360:
    set_motion_accelonly();
361:
    set_motion_busy();
362:
    set_motion_decelonly();
363:
    set_motion_index_dist();
364:
    set_motion_index_num();
365:
    set_motion_tracking_ai();
366:
    set_motion_tracking_dir();
367:
    set_motion_tracking_ki();
368:
    set_motion_tracking_kp();
369:
    set_motion_tracking_limit_max();
370:
    set_motion_tracking_limit_min();
371:
    set_motion_tracking_scan_dir();
372:
    set_motion_tracking_scan_maxspeed();
373:
    set_motion_tracking_scan_offset();
374:
    set_motion_tracking_scan_period();
375:
    set_motion_tracking_scan_signal_valid_delay();
376:
    set_motion_tracking_scan_tolerance();
377:
    set_motion_tracking_setpoint();
378:
    set_motion_tracking_settle_period();
379:
    set_motion_tracking_settle_tolerance();
380:
    set_motion_tracking_settle_tolerance_met();
381:
    set_motion_tracking_settled();
382:
    set_motion_tracking_signal_valid_di();
383:
    set_motor_current_max();
384:
    set_motor_inductance();
385:
    set_motor_ke();
386:
    set_motor_phase();
387:
    set_motor_phase_ratio_div1();
388:
    set_motor_phase_ratio_div2();
389:
    set_motor_phase_ratio_mult();
390:
    set_motor_resistance();
391:
    set_parking_state();
392:
    set_peripheral_hw_modified();
393:
    set_peripheral_id();
394:
    set_peripheral_id_pending();
395:
    set_peripheral_serial();
396:
    set_peripheral_serial_pending();
397:
    set_pos();
398:
    set_pvt_numseqs();
399:
    set_resolution();
400:
    set_scope_channel_size();
401:
    set_scope_channel_size_max();
402:
    set_scope_delay();
403:
    set_scope_numchannels();
404:
    set_scope_timebase();
405:
    set_stream_numbufs();
406:
    set_stream_numstreams();
407:
    set_system_access();
408:
    set_system_axiscount();
409:
    set_system_led_enable();
410:
    set_system_serial();
411:
    set_system_temperature();
412:
    set_system_uptime();
413:
    set_system_voltage();
414:
    set_trigger_numactions();
415:
    set_trigger_numtriggers();
416:
    set_user_data_0();
417:
    set_user_data_1();
418:
    set_user_data_2();
419:
    set_user_data_3();
420:
    set_user_data_4();
421:
    set_user_data_5();
422:
    set_user_data_6();
423:
    set_user_data_7();
424:
    set_user_data_8();
425:
    set_user_data_9();
426:
    set_user_data_10();
427:
    set_user_data_11();
428:
    set_user_data_12();
429:
    set_user_data_13();
430:
    set_user_data_14();
431:
    set_user_data_15();
432:
    set_user_vdata_0();
433:
    set_user_vdata_1();
434:
    set_user_vdata_2();
435:
    set_user_vdata_3();
436:
    set_vel();
437:
    set_version();
438:
    set_version_build();
439:
	warnings_clear();
END_CASE
END_METHOD

METHOD PROTECTED _MonitorAsynchronousRequests
//FIFO this
// IF WaitingForBits.WaitingForResolution THEN
// 	ZaberConfiguration.Resolution := STRING_TO_REAL(F_GetFirstWordInString(sInput := ZaberStatus.ZaberReply.DataField));
// 	WaitingForBits.WaitingForResolution	:= FALSE;
// END_IF

IF WaitingForBits.WaitingForMaxSpeed THEN
	ZaberStatus.Velocity := STRING_TO_DINT(F_GetFirstWordInString(sInput := ZaberStatus.ZaberReply.DataField));
	WaitingForBits.WaitingForMaxSpeed 	:= FALSE;
END_IF
END_METHOD

METHOD PROTECTED _PollBusy
IF ZaberStatus.NewResponseParsed THEN
	PollBusyTimer.IN := TRUE;
END_IF

IF PollBusyTimer.Q THEN
	//get_motion_busy();
	get_pos();
	//get_vel();
	PollBusyTimer.IN := FALSE; // One-shot until BUSY is confirmed again
END_IF

IF ZaberConfiguration.EnableDynamicPollingInterval AND_THEN (ZaberStatus.Velocity <> 0) AND (ZaberConfiguration.SetDynamics.Velocity <> 0) THEN
ZaberConfiguration.PollingIntervalTime := 
    LREAL_TO_TIME(
        Base.F_MapLREAL(
            in_max := (1000 * ZaberConfiguration.Resolution_um), // 1 step resolution
            in_min := 1000 * (ZaberConfiguration.Resolution_um / (ABS(ZaberConfiguration.SetDynamics.Velocity))),
            out_max := TIME_TO_LREAL(ZaberConfiguration.MaxPollingTime),
            out_min := TIME_TO_LREAL(ZaberConfiguration.MinPollingTime),
            x := 1000 * (ZaberConfiguration.Resolution_um / DINT_TO_REAL(ABS(ZaberStatus.Velocity)))
        )
    );
ELSE
	ZaberConfiguration.PollingIntervalTime := ZaberConfiguration.DefaultPollingTime;
END_IF

PollBusyTimer(PT := ZaberConfiguration.PollingIntervalTime);
END_METHOD

METHOD PROTECTED _PopulateStatusStructureWithResponseData
ZaberStatus.ZaberReply.DeviceAddress	:= F_ExtractDeviceAddress(iBufferRcv.P_LastObjectRead.stringval);
ZaberStatus.ZaberReply.AxisNumber		:= F_ExtractAxisNumber(iBufferRcv.P_LastObjectRead.stringval);
ZaberStatus.ZaberReply.WarnFlag       	:= F_ZaberExtractWarnFaultFlag(iBufferRcv.P_LastObjectRead.stringval);
ZaberStatus.ZaberReply.ReplyFlag   		:= F_ZaberExtractExecutionResult(iBufferRcv.P_LastObjectRead.stringval);
ZaberStatus.ZaberReply.MotionStatus		:= F_ExtractMotionStatus(iBufferRcv.P_LastObjectRead.stringval);
ZaberStatus.ZaberReply.DataField		:= F_ExtractDataField(iBufferRcv.P_LastObjectRead.stringval);

IF ZaberStatus.ZaberReply.ReplyFlag = 'RJ' THEN
	TraceWithSeverity(Message := CONCAT('Zaber Axis Command Rejected; Reason: ', ZaberStatus.ZaberReply.DataField), Severity := TcEventSeverity.Warning);
END_IF

IF ZaberStatus.ZaberReply.WarnFlag <> '--' THEN
    TraceWithSeverity(Message := CONCAT('Zaber Axis Warning/Fault: ', ZaberStatus.ZaberReply.WarnFlag), Severity := TcEventSeverity.Warning);
END_IF

IF ZaberStatus.ZaberReply.ReplyFlag = 'RJ' AND (F_ZaberExtractExecutionResult(ZaberStatus.ZaberReply.DataField) <> '') THEN
	TraceWithSeverity(Message := CONCAT('Zaber Axis Error: ', ZaberStatus.ZaberReply.DataField), Severity := TcEventSeverity.Error);
END_IF

CASE ZaberStatus.ZaberMethodDispatch OF

242:
	ZaberStatus.Position		:= ABS(STRING_TO_DINT(F_GetFirstWordInString(ZaberStatus.ZaberReply.DataField)));
282:	
	ZaberStatus.Velocity		:= ABS(STRING_TO_DINT(F_GetFirstWordInString(ZaberStatus.ZaberReply.DataField)));

END_CASE
ZaberStatus.ZaberReply.Checksum			:= F_ExtractMessageChecksum(iBufferRcv.P_LastObjectRead.stringval);
END_METHOD

METHOD PROTECTED _ReceiveCyclic
VAR_INST
	ControllerString : STRING;
	AxisString : STRING;
END_VAR
IF _iSerialRx <> 0 AND iBufferRcv <> 0 AND iBufferAll <> 0 THEN
	IF _iSerialRx.P_ReceiveStringStatus.bStringReceived THEN
		//Confirm the message received is addressed to this instance
		ControllerString	:= Tc2_Standard.RIGHT(STR := Base.F_GetFirstWordInString(_iSerialRx.P_ReceiveStringStatus.StringRx.sCurrentStringFormatted), SIZE := 1);
		AxisString := Tc2_Standard.LEFT(STR := F_GetAllButFirstWord(sInput := _iSerialRx.P_ReceiveStringStatus.StringRx.sCurrentStringFormatted), SIZE := 1);
	// 	IF (ControllerString = Tc2_Standard.RIGHT(STR := _ZaberSerialConfiguration.P_ZaberConfiguration.sControllerRef, SIZE := 1)) AND
	//	IF (AxisString = UINT_TO_STRING(_ZaberSerialConfiguration.P_ZaberConfiguration.AxisRef)) THEN
			ZaberReceipt.stringval	:= _iSerialRx.P_ReceiveStringStatus.StringRx.sCurrentStringFormatted;
			iBufferRcv.AddObject(RefObject := ZaberReceipt);
			iBufferAll.AddObject(RefObject := ZaberReceipt);
	//	END_IF
	END_IF
END_IF

IF iBufferRcv <> 0 THEN
	IF iBufferRcv.P_ObjectWasAdded THEN
		iBufferRcv.ReadObject();
		iBufferRcv.ClearStatusFlagAdded();
	END_IF
	
	//Parse the received string to struct
	IF iBufferRcv.P_ObjectWasRead THEN
		
		_PopulateStatusStructureWithResponseData();
		
		_MonitorAsynchronousRequests();
		
		iBufferRcv.ClearStatusFlagRead();
		ZaberStatus.NewResponseParsed  		:= TRUE;
	ELSE
		ZaberStatus.NewResponseParsed  		:= FALSE;
	END_IF
END_IF
END_METHOD

METHOD PRIVATE _ResolveZaberConfiguration : REFERENCE TO ST_ZaberConfiguration
IF _ZaberSerialConfiguration <> 0 THEN
	_ResolveZaberConfiguration	REF= _ZaberSerialConfiguration.P_ZaberConfiguration;
	ZaberConfiguration := _ResolveZaberConfiguration;
	ZaberStatus.ConfigurationResolution	:= E_ConfigurationResolution.InjectedInterface;
ELSE
	_ResolveZaberConfiguration	REF= ZaberConfiguration;
	//ZaberStatus.ConfigurationResolution	:= E_ConfigurationResolution.Local;
	TraceWithSeverity(Message := 'Using Local Zaber Configuration - pass interface', Severity := TcEventSeverity.Info);
END_IF
END_METHOD

METHOD PROTECTED _ResolveZaberDispatchIndex : DINT
VAR_INPUT
	sPOUName 		: STRING;
END_VAR
VAR
	idx 			: DINT;
	bResolved		: BOOL := FALSE;
END_VAR
FOR idx := GC_Zaber.INDEX_COMMAND_MIN TO GC_Zaber.INDEX_COMMAND_MAX DO
	IF sPOUName = SUPER^._iCommandConfiguration[idx].P_CommandConfiguration.CommandPOUName THEN
		_ResolveZaberDispatchIndex := idx;
		bResolved := TRUE;
		EXIT;
	END_IF
END_FOR

IF NOT bResolved THEN
	_ResolveZaberDispatchIndex := -1;

	IF ZaberConfiguration.ComponentConfiguration.BaseConfiguration.LogTraceConfiguration.What.xLogToEventLogger AND 
	   ZaberConfiguration.ComponentConfiguration.BaseConfiguration.LogTraceConfiguration.When = E_LogTraceWhen.xRunCyclic THEN
		TraceWithSeverity(Message := Tc2_Standard.CONCAT(STR1 := 'Invalid POU name commanded: ', STR2 := sPOUName), Severity := TcEventSeverity.Error);
	END_IF
END_IF
END_METHOD

METHOD PROTECTED _SendCyclic
IF iBufferSend <> 0 AND iBufferAll <> 0 THEN
	IF iBufferSend.P_ObjectWasAdded THEN
		iBufferSend.ReadObject();
		iBufferSend.ClearStatusFlagAdded();
	END_IF
	
	IF iBufferSend.P_ObjectWasRead THEN
		iBufferAll.AddObject(RefObject := iBufferSend.P_LastObjectRead);
		_iSerialTx.SendString(StringToSend := iBufferSend.P_LastObjectRead.stringval);
		//TraceWithSeverity(Message := CONCAT(STR1 := iBufferSend.P_LastObjectRead.stringval, STR2 := ULINT_TO_STRING(iBufferSend.P_LastObjectRead.systimestamp)), Severity := TcEventSeverity.Info);
		iBufferSend.ClearStatusFlagRead();
	END_IF
END_IF
END_METHOD

METHOD PROTECTED _TryRehashDispatchIndex : BOOL
VAR_INPUT
    sCommandPOUName : STRING;
END_VAR
IF _ZaberAxisConfigurationFW744 = 0 THEN
    TraceWithSeverity('Hash table is NULL � command aborted', TcEventSeverity.Error);
    _TryRehashDispatchIndex := FALSE;
    RETURN;
END_IF

//Rehash
ZaberStatus.ZaberMethodDispatch := _ZaberAxisConfigurationFW744.GetIndexByPOUName(NameIn := sCommandPOUName);

IF NOT ((ZaberStatus.ZaberMethodDispatch >= LOWER_BOUND(SUPER^.Commands, 1)) AND
        (ZaberStatus.ZaberMethodDispatch <= UPPER_BOUND(SUPER^.Commands, 1))) THEN
    	TraceWithSeverity('Hashing failed.  Interface valid but hash table may have no initial insert', TcEventSeverity.Error);

    _TryRehashDispatchIndex := FALSE;
    RETURN;
END_IF

_TryRehashDispatchIndex := TRUE;
END_METHOD

(*override for continuous execution use
example code

// Base implementation - Component derivatives should override this method
// This method maps from command index to business logic method calls
// Called from _CommandsCyclic when Commands[CommandIndex] is busy

CASE ComponentStatus.iLastCommandConfiguration.P_CommandConfiguration.CommandIndex OF

MinIndexComponentCmd..MaxIndexComponentCmd:
	// Valid command index range
	// Component derivatives should override this method to handle specific command indices
	// Example pattern from FB_FileHandlerCsv:
	// 
	// GC_FILE.INDEX_OPENFILE:
	//     _OpenFile();
	// 
	// GC_FILE.INDEX_CLOSEFILE:
	//     _CloseFile();
	
	// Base class: No specific implementation - just a placeholder

ELSE
	// Invalid index - trace error
	IF SUPER^.BaseConfiguration.LogTraceConfiguration.What.xLogToEventLogger THEN
		TraceWithSeverity(Message := 'Invalid CommandIndex in _ExecuteCommandByIndex', Severity := Global.TcEventSeverity.Warning);
	END_IF
END_CASE;

*)
METHOD PROTECTED _ExecuteCommandByIndexCyclic
END_METHOD

METHOD ExecuteCommand : Base.I_ComponentFull
VAR_INPUT
	CmdIndex	: DINT;
END_VAR
IF CmdIndex >= LOWER_BOUND(SUPER^.Commands,1) AND CmdIndex <= UPPER_BOUND(SUPER^.Commands,1) THEN
	SUPER^.ExecuteCommand(CmdIndex := CmdIndex);
	
	IF SUPER^.iCommands[CmdIndex].P_CommandStatus.Result = Base.E_HttpStatusCode.Ok THEN
		ZaberStatus.ZaberMethodDispatch	:= CmdIndex;
	END_IF
	
	_MapIndicesToCommands();
ELSE
	TraceWithSeverity(Message := Tc2_Standard.CONCAT(STR1 := DINT_TO_STRING(CmdIndex), STR2 := ' not within array bounds'), Severity := TcEventSeverity.Error);
END_IF

ExecuteCommand := THIS^;
END_METHOD

METHOD InjectConfigurations
VAR_INPUT
	CommandConfigurations		: ARRAY[GC_Zaber.INDEX_COMMAND_MIN..GC_Zaber.INDEX_COMMAND_MAX] OF I_CommandConfiguration;	
	PermIntlkConfigurations		: ARRAY[GC_Zaber.INDEX_COMMAND_MIN..GC_Zaber.INDEX_COMMAND_MAX] OF I_PermIntlkConfiguration;
	AxisConfiguration			: I_ZaberAxisConfigurationFW744; //MAY obviate the other arrays^
	AxisSerialConfiguration		: I_ZaberSerialConfiguration;
END_VAR
FOR SUPER^.CommandIndexCyclic := LOWER_BOUND(SUPER^.Commands, 1) TO UPPER_BOUND(SUPER^.Commands, 1) DO
    IF (CommandConfigurations[SUPER^.CommandIndexCyclic] <> 0) AND 
       (PermIntlkConfigurations[SUPER^.CommandIndexCyclic] <> 0) THEN
	   
		SUPER^._iCommandConfiguration[SUPER^.CommandIndexCyclic]	:= CommandConfigurations[SUPER^.CommandIndexCyclic];
		SUPER^._iPermIntlkConfiguration[SUPER^.CommandIndexCyclic]	:= PermIntlkConfigurations[SUPER^.CommandIndexCyclic];
		
		SUPER^.Commands[SUPER^.CommandIndexCyclic].InjectConfigurations(iComponent := THIS^, iCommandConfiguration := CommandConfigurations[SUPER^.CommandIndexCyclic], 
																		iPermIntlkConfiguration := PermIntlkConfigurations[SUPER^.CommandIndexCyclic]);

    ELSIF (CommandConfigurations[SUPER^.CommandIndexCyclic] = 0) THEN 
        IF ZaberConfiguration.ComponentConfiguration.BaseConfiguration.LogTraceConfiguration.What.xLogToEventLogger THEN
			TraceWithSeverity(Message := CONCAT('Command Configuration interface not provided at index ', DINT_TO_STRING(SUPER^.CommandIndexCyclic)), Severity := TcEventSeverity.Error);
		END_IF
	ELSIF (PermIntlkConfigurations[SUPER^.CommandIndexCyclic] = 0) THEN 
        IF ZaberConfiguration.ComponentConfiguration.BaseConfiguration.LogTraceConfiguration.What.xLogToEventLogger THEN
			TraceWithSeverity(Message := CONCAT('PermIntlk Configuration interface not provided at index ', DINT_TO_STRING(SUPER^.CommandIndexCyclic)), Severity := TcEventSeverity.Error);
		END_IF
    END_IF
END_FOR

_ZaberAxisConfigurationFW744 := AxisConfiguration;
_ZaberSerialConfiguration	:= AxisSerialConfiguration;
END_METHOD

PROPERTY P_I_RingBufferKeyString : REFERENCE TO Base.I_RingBufferKeyString
GET
IF iBufferAll <> 0 THEN
	P_I_RingBufferKeyString REF= iBufferAll;
END_IF
END_GET
END_PROPERTY

END_FUNCTION_BLOCK

// Zaber/POUs/FB_ZaberSerialGroup
FUNCTION_BLOCK FB_ZaberSerialGroup EXTENDS Base.FB_BaseCyclic
VAR
	DeskTesting 						: BOOL := TRUE;
	
//System
//	ControlMode							: Base.FB_ControlMode();
	iControlMode						: Base.I_ControlMode; // := ControlMode;
// 	SysPermIntlk						: Base.FB_PermIntlk();
	iSysPermIntlk						: Base.I_PermIntlk; // := SysPermIntlk;
	                            		
//Serial Interface              		
	SerialCommunication					: Communication.FB_Serial;
	iSerialConfig						: Communication.I_SerialConfiguration := SerialCommunication;
	iSerialComm							: Communication.I_SerialStatus := SerialCommunication;
	iSerialTx							: Communication.I_StringCmdStatusTx := SerialCommunication;
	iSerialRx							: Communication.I_StringCmdStatusRx := SerialCommunication;

//Configuration
	ZaberConfigurations					: ARRAY[GPL_Zaber.INDEX_AXISGRPINST_MIN..GPL_Zaber.INDEX_AXISGRPINST_MAX] OF FB_ZaberAxisCmdConfiguration;
	iZaberCmdConfigurations				: ARRAY[GPL_Zaber.INDEX_AXISGRPINST_MIN..GPL_Zaber.INDEX_AXISGRPINST_MAX] OF I_ZaberAxisConfigurationFW744; //ZaberConfigurations
	iZaberAxisConfigurations			: ARRAY[GPL_Zaber.INDEX_AXISGRPINST_MIN..GPL_Zaber.INDEX_AXISGRPINST_MAX] OF I_ZaberSerialConfiguration; //ZaberConfigurations
	                            		
	ZaberAxes							: ARRAY[GPL_Zaber.INDEX_AXISGRPINST_MIN..GPL_Zaber.INDEX_AXISGRPINST_MAX] OF FB_ZaberSerialAxis;
	iZaberAxes							: ARRAY[GPL_Zaber.INDEX_AXISGRPINST_MIN..GPL_Zaber.INDEX_AXISGRPINST_MAX] OF I_ZaberSerialFW744; //ZaberAxes
	iZaberComponents					: ARRAY[GPL_Zaber.INDEX_AXISGRPINST_MIN..GPL_Zaber.INDEX_AXISGRPINST_MAX] OF Base.I_ComponentFull; //ZaberAxes

	LoopIndex							: DINT;
	
	SelectedAxisIndex					: DINT := 1;

	DebugString							: STRING;
	stDebugStrings						: ST_ZaberInitTableFW744;
	RingBufferDebugString				: Base.FB_RingBufferString;
	iRingBufferString					: Base.I_RingBufferString := RingBufferDebugString;
	RingBufferDebugUint					: Base.FB_RingBufferUINT;
	iRingBufferDebugUint				: Base.I_RingBufferUINT := RingBufferDebugUint;

//Test Triggers
 	TriggerAllCommands					: BOOL;
	TrigIntervalTime					: TIME := T#200MS;
	TrigIntervalTimer					: Tc2_Standard.TON;
	TrigIndex							: DINT;

//Debug State Machine
	CurrTrigIndex 						: DINT := GPL_Zaber.INDEX_COMMAND_MIN;
	State         						: INT := 0; // 0 = Idle, 1 = Wait, 2 = Advance
	SequenceActive						: BOOL;

//File Operations
// 	FileHandlerCsv						: FB_FileHandlerCsv;
// 	iFileHandlerCsv						: I_FileHandlerCsv := FileHandlerCsv;
	TempCountObjectsToWrite				: UDINT;
	TempRingObj							: Base.ST_SystimeString;
	TempUint							: UINT;
	i									: DINT;
	TrigOpenFile						: BOOL;
	TrigCloseFile						: BOOL;
	TrigWriteToFile						: BOOL;
	TrigWriteIndicesToFile				: BOOL;
	
	TrigStopAll							: BOOL;
END_VAR

METHOD PRIVATE _ControllerAxisConfiguration
//Setting Configurations

// IF iZaberAxisConfigurations[0] <> 0 (*AND __QUERYINTERFACE()*) THEN
// 	iZaberAxisConfigurations[0].P_ZaberConfiguration.sControllerRef := '/1';
// 	iZaberAxisConfigurations[0].P_ZaberConfiguration.AxisRef		:= 1;
// END_IF


IF iZaberAxisConfigurations[1] <> 0 (*AND __QUERYINTERFACE()*) THEN
	IF DeskTesting THEN
		iZaberAxisConfigurations[1].P_ZaberConfiguration.sControllerRef := '/0';
		iZaberAxisConfigurations[1].P_ZaberConfiguration.AxisRef		:= 0;
	ELSE
		iZaberAxisConfigurations[1].P_ZaberConfiguration.sControllerRef := '/1';
		iZaberAxisConfigurations[1].P_ZaberConfiguration.AxisRef		:= 2;
		iZaberAxisConfigurations[1].P_ZaberConfiguration.LockstepGroup	:= 1;
	END_IF
END_IF

// 
// IF iZaberAxisConfigurations[2] <> 0 (*AND __QUERYINTERFACE()*) THEN
// 	iZaberAxisConfigurations[2].P_ZaberConfiguration.sControllerRef := '/2';
// 	iZaberAxisConfigurations[2].P_ZaberConfiguration.AxisRef		:= 1;
// 	iZaberAxisConfigurations[2].P_ZaberConfiguration.LockstepGroup	:= 1;
// END_IF
// 
// 
// IF iZaberAxisConfigurations[3] <> 0 (*AND __QUERYINTERFACE()*) THEN
// 	iZaberAxisConfigurations[3].P_ZaberConfiguration.sControllerRef := '/2';
// 	iZaberAxisConfigurations[3].P_ZaberConfiguration.AxisRef		:= 3;
// 	iZaberAxisConfigurations[3].P_ZaberConfiguration.LockstepGroup	:= 2;
// END_IF
// 
// IF iZaberAxisConfigurations[4] <> 0 (*AND __QUERYINTERFACE()*) THEN
// 	iZaberAxisConfigurations[4].P_ZaberConfiguration.sControllerRef := '/3';
// 	iZaberAxisConfigurations[4].P_ZaberConfiguration.AxisRef		:= 1;
// END_IF
// 
// 
// IF iZaberAxisConfigurations[5] <> 0 (*AND __QUERYINTERFACE()*) THEN
// 	iZaberAxisConfigurations[5].P_ZaberConfiguration.sControllerRef := '/3';
// 	iZaberAxisConfigurations[5].P_ZaberConfiguration.AxisRef		:= 2;
// END_IF
// 
// 
// IF iZaberAxisConfigurations[6] <> 0 (*AND __QUERYINTERFACE()*) THEN
// 	iZaberAxisConfigurations[6].P_ZaberConfiguration.sControllerRef := '/4';
// 	iZaberAxisConfigurations[6].P_ZaberConfiguration.AxisRef		:= 0;
// END_IF
//
END_METHOD

(* Basic component initialization logic*)
METHOD PROTECTED _Initialize : BOOL
BaseStatus.Initialized := _InitializeChildrenDependencies();

BaseStatus.Initialized	:= _InitializeReferences();

BaseStatus.Busy	:= FALSE;

IF NOT BaseStatus.Initialized THEN
	TraceWithSeverity(Message := 'Initialization Failed - look at _Initialize method', Severity := TcEventSeverity.Error);
END_IF
								
FOR LoopIndex := LOWER_BOUND(ZaberAxes,1) TO UPPER_BOUND(ZaberAxes,1) BY 1 DO
// Injection
	ZaberAxes[LoopIndex].InjectConfigurations(CommandConfigurations := iZaberCmdConfigurations[LoopIndex].P_CommandConfigurations, 
								PermIntlkConfigurations := iZaberCmdConfigurations[LoopIndex].P_PermIntlkConfigurations,
								AxisConfiguration := iZaberCmdConfigurations[LoopIndex],
								AxisSerialConfiguration := iZaberAxisConfigurations[LoopIndex]);
END_FOR

_ControllerAxisConfiguration();

_Initialize 	:= TRUE;
END_METHOD

METHOD PROTECTED _InitializeChildrenDependencies : BOOL
// ControlMode.Initialize();
// 
// SysPermIntlk.Initialize();

SerialCommunication.Initialize();

FOR LoopIndex := LOWER_BOUND(ZaberAxes,1) TO UPPER_BOUND(ZaberAxes,1) BY 1 DO
	ZaberConfigurations[LoopIndex].Initialize();
	ZaberAxes[LoopIndex].Initialize();
END_FOR

RingBufferDebugString.Initialize();

RingBufferDebugUint.Initialize();

// FileHandlerCsv.Initialize();

_InitializeChildrenDependencies := TRUE;
END_METHOD

METHOD CyclicLogic
SUPER^.CyclicLogic();

IF iSerialComm <> 0 THEN
	iSerialComm.CyclicLogic();
END_IF

FOR LoopIndex := LOWER_BOUND(ZaberAxes,1) TO UPPER_BOUND(ZaberAxes,1) BY 1 DO

	ZaberAxes[LoopIndex].CyclicLogic();
	
	IF TrigStopAll THEN
		ZaberAxes[LoopIndex].stop();
		TrigStopAll	:= FALSE;
	END_IF
END_FOR

//--------------------------
// Debug State Machine - Runs through all commands on the Controller with an interval time between commands
//--------------------------

CASE State OF

    0: // Idle - wait for start trigger
        IF TriggerAllCommands THEN
			SequenceActive := TRUE;
			CurrTrigIndex := GPL_Zaber.INDEX_COMMAND_MIN;
			TriggerAllCommands := FALSE; // reset trigger
		END_IF

		IF SequenceActive THEN
			IF iZaberComponents[SelectedAxisIndex] <> 0 THEN
				iZaberComponents[SelectedAxisIndex].ExecuteCommand(CmdIndex := CurrTrigIndex);
				TrigIntervalTimer.IN := TRUE;
				State := 1;
			END_IF
        END_IF

    1: // Wait for interval after command
        IF TrigIntervalTimer.Q THEN
            TrigIntervalTimer.IN := FALSE;

            CurrTrigIndex := CurrTrigIndex + 1;

            IF CurrTrigIndex <= GPL_Zaber.INDEX_COMMAND_MAX THEN
                State := 0;
                // stay in state 1
            ELSE
                SequenceActive := FALSE;
                State := 0;
            END_IF
        END_IF

END_CASE

TrigIntervalTimer(PT := TrigIntervalTime);

//--------------------------
// File Operations
//--------------------------
// iFileHandlerCsv.CyclicLogic();
// 
// IF TrigOpenFile THEN
// 	iFileHandlerCsv.OpenFile();
// 	TrigOpenFile	:= FALSE;
// END_IF

// IF TrigWriteToFile THEN
// 	IF ZaberAxes[SelectedAxisIndex].P_I_RingBufferKeyString <> 0 THEN
// 		TempCountObjectsToWrite	:= 0;
// 		TempCountObjectsToWrite := ZaberAxes[SelectedAxisIndex].P_I_RingBufferKeyString.P_RingBufferStatus.ObjectCountInBufferPrim - 1;
// 
// 		FOR i := LOWER_BOUND(ZaberAxes[SelectedAxisIndex].P_I_RingBufferKeyString.P_Buffer,1) TO UPPER_BOUND(ZaberAxes[SelectedAxisIndex].P_I_RingBufferKeyString.P_Buffer,1) DO
// 			TempRingObj := ZaberAxes[SelectedAxisIndex].P_I_RingBufferKeyString.P_Buffer[i];
// 
// 			IF (TempRingObj.systimestamp <> 0) OR (LEN(TempRingObj.stringval) > 0) THEN
// 				// Append field
// 				iFileHandlerCsv.AppendToFileBySystimeString(sContent := TempRingObj);
// 			END_IF
// 		END_FOR
// 
// 	END_IF
// 	TrigWriteToFile := FALSE;
// END_IF

// IF TrigWriteIndicesToFile THEN
// 	FOR i := LOWER_BOUND(stDebugStrings.aDebugStrings,1) TO UPPER_BOUND(stDebugStrings.aDebugStrings,1) DO
// 		IF iRingBufferDebugUint <> 0 THEN
// 			TempUint := iRingBufferDebugUint.P_Buffer[i];
// 		END_IF
// 
// 		// Append field
// 		IF iFileHandlerCsv <> 0 THEN
// 			iFileHandlerCsv.AppendToFileByString(sContent := UINT_TO_STRING(TempUint));
// 		END_IF
// 		
//     END_FOR
// 	TrigWriteIndicesToFile	:= FALSE;
// END_IF
// 
// IF TrigCloseFile AND (iFileHandlerCsv.P_FileHandlerCsvStatus.FileHandle <> 0) AND (iFileHandlerCsv.P_AppendRingBufferStatus.ObjectCountInBufferPrim = 0) THEN 
// 	iFileHandlerCsv.CloseFile();
// 	TrigCloseFile	:= FALSE;
// END_IF
END_METHOD

//FB_Init is always available implicitly and it is used primarily for initialization.
//The return value is not evaluated. For a specific influence, you can also declare the
//methods explicitly and provide additional code there with the standard initialization
//code. You can evaluate the return value.
METHOD FB_Init: BOOL
VAR_INPUT
    bInitRetains: BOOL; // TRUE: the retain variables are initialized (reset warm / reset cold)
    bInCopyCode: BOOL;  // TRUE: the instance will be copied to the copy code afterward (online change)   
END_VAR
FOR LoopIndex := LOWER_BOUND(ZaberAxes,1) TO UPPER_BOUND(ZaberAxes,1) BY 1 DO
	//Wiring
	iZaberCmdConfigurations[LoopIndex]	:= ZaberConfigurations[LoopIndex];
	iZaberAxisConfigurations[LoopIndex]	:= ZaberConfigurations[LoopIndex];
	iZaberAxes[LoopIndex]				:= ZaberAxes[LoopIndex];
	iZaberComponents[LoopIndex]			:= ZaberAxes[LoopIndex];
END_FOR
END_METHOD

END_FUNCTION_BLOCK

// Zaber/Testing/FB_ValidateStringHandlingTests
FUNCTION_BLOCK FB_ValidateStringHandlingTests EXTENDS TcUnit.FB_TestSuite

GivenBusyReplyExpectCorrectFieldExtractionChecksum();
GivenBusyReplyExpectCorrectFieldExtractionNoChecksum();
GivenIdleReplyExpectCorrectFieldExtractionChecksum();
GivenIdleReplyExpectCorrectFieldExtractionNoChecksum();
GivenNIReplyExpectCorrectFieldExtractionChecksum();
GivenNIReplyExpectCorrectFieldExtractionNoChecksum();
GivenReply_ExpectCorrectTokenization();
GivenIdleReplyExpectCorrectFieldExtractionChecksum_1();

METHOD PRIVATE GivenBusyReplyExpectCorrectFieldExtractionChecksum
VAR
    InputReply         : STRING := '@02 0 OK BUSY -- -15000 NA:C5';
    ExpectedAddress    : STRING := '02';
    ExpectedAxis       : STRING := '0';
    ExpectedResult     : STRING := 'OK';
    ExpectedMotion     : STRING := 'BUSY';
    ExpectedWarnFault  : STRING := '--';
    ExpectedDataField  : STRING := '-15000 NA';
    ExpectedChecksum   : STRING := 'C5';

    ActualAddress      : STRING;
    ActualAxis         : STRING;
    ActualResult       : STRING;
    ActualMotion       : STRING;
    ActualWarnFault    : STRING;
    ActualDataField    : STRING;
    ActualChecksum     : STRING;
END_VAR
TEST(__POUNAME());

// Execute field extraction
ActualAddress     := F_ExtractDeviceAddress(sInput := InputReply);
ActualAxis        := F_ExtractAxisNumber(sInput := InputReply);
ActualResult      := F_ZaberExtractExecutionResult(sInput := InputReply);
ActualMotion      := F_ExtractMotionStatus(sInput := InputReply);
ActualWarnFault   := F_ZaberExtractWarnFaultFlag(sInput := InputReply);
ActualDataField   := F_ExtractDataField(sInput := InputReply);
ActualChecksum    := F_ExtractMessageChecksum(sInput := InputReply);

// Assertions
AssertEquals(Expected := ExpectedAddress, Actual := ActualAddress, Message := 'Device Address mismatch');
AssertEquals(Expected := ExpectedAxis, Actual := ActualAxis, Message := 'Axis Number mismatch');
AssertEquals(Expected := ExpectedResult, Actual := ActualResult, Message := 'Execution Result mismatch');
AssertEquals(Expected := ExpectedMotion, Actual := ActualMotion, Message := 'Motion Status mismatch');
AssertEquals(Expected := ExpectedWarnFault, Actual := ActualWarnFault, Message := 'Warning/Fault Flag mismatch');
AssertEquals(Expected := ExpectedDataField, Actual := ActualDataField, Message := 'Data Field mismatch');
AssertEquals(Expected := ExpectedChecksum, Actual := ActualChecksum, Message := 'Checksum mismatch');

TEST_FINISHED();
END_METHOD

METHOD PRIVATE GivenBusyReplyExpectCorrectFieldExtractionNoChecksum
VAR
    InputReply         : STRING := '@02 0 OK BUSY -- -15000 NA';
    ExpectedAddress    : STRING := '02';
    ExpectedAxis       : STRING := '0';
    ExpectedResult     : STRING := 'OK';
    ExpectedMotion     : STRING := 'BUSY';
    ExpectedWarnFault  : STRING := '--';
    ExpectedDataField  : STRING := '-15000 NA';
    ExpectedChecksum   : STRING := '';

    ActualAddress      : STRING;
    ActualAxis         : STRING;
    ActualResult       : STRING;
    ActualMotion       : STRING;
    ActualWarnFault    : STRING;
    ActualDataField    : STRING;
    ActualChecksum     : STRING;
END_VAR
TEST(__POUNAME());

// Execute field extraction
ActualAddress     := F_ExtractDeviceAddress(sInput := InputReply);
ActualAxis        := F_ExtractAxisNumber(sInput := InputReply);
ActualResult      := F_ZaberExtractExecutionResult(sInput := InputReply);
ActualMotion      := F_ExtractMotionStatus(sInput := InputReply);
ActualWarnFault   := F_ZaberExtractWarnFaultFlag(sInput := InputReply);
ActualDataField   := F_ExtractDataField(sInput := InputReply);
ActualChecksum    := F_ExtractMessageChecksum(sInput := InputReply);

// Assertions
AssertEquals(Expected := ExpectedAddress, Actual := ActualAddress, Message := 'Device Address mismatch');
AssertEquals(Expected := ExpectedAxis, Actual := ActualAxis, Message := 'Axis Number mismatch');
AssertEquals(Expected := ExpectedResult, Actual := ActualResult, Message := 'Execution Result mismatch');
AssertEquals(Expected := ExpectedMotion, Actual := ActualMotion, Message := 'Motion Status mismatch');
AssertEquals(Expected := ExpectedWarnFault, Actual := ActualWarnFault, Message := 'Warning/Fault Flag mismatch');
AssertEquals(Expected := ExpectedDataField, Actual := ActualDataField, Message := 'Data Field mismatch');
AssertEquals(Expected := ExpectedChecksum, Actual := ActualChecksum, Message := 'Checksum mismatch');

TEST_FINISHED();
END_METHOD

METHOD PRIVATE GivenIdleReplyExpectCorrectFieldExtractionChecksum
VAR
    InputReply         : STRING := '@02 0 OK IDLE -- 0 NA:DD';
    ExpectedAddress    : STRING := '02';
    ExpectedAxis       : STRING := '0';
    ExpectedResult     : STRING := 'OK';
    ExpectedMotion     : STRING := 'IDLE';
    ExpectedWarnFault  : STRING := '--';
    ExpectedDataField  : STRING := '0 NA';
    ExpectedChecksum   : STRING := 'DD';

    ActualAddress      : STRING;
    ActualAxis         : STRING;
    ActualResult       : STRING;
    ActualMotion       : STRING;
    ActualWarnFault    : STRING;
    ActualDataField    : STRING;
    ActualChecksum     : STRING;
END_VAR
TEST(__POUNAME());

// Execute field extraction
ActualAddress     := F_ExtractDeviceAddress(sInput := InputReply);
ActualAxis        := F_ExtractAxisNumber(sInput := InputReply);
ActualResult      := F_ZaberExtractExecutionResult(sInput := InputReply);
ActualMotion      := F_ExtractMotionStatus(sInput := InputReply);
ActualWarnFault   := F_ZaberExtractWarnFaultFlag(sInput := InputReply);
ActualDataField   := F_ExtractDataField(sInput := InputReply);
ActualChecksum    := F_ExtractMessageChecksum(sInput := InputReply);

// Assertions
AssertEquals(Expected := ExpectedAddress, Actual := ActualAddress, Message := 'Device Address mismatch');
AssertEquals(Expected := ExpectedAxis, Actual := ActualAxis, Message := 'Axis Number mismatch');
AssertEquals(Expected := ExpectedResult, Actual := ActualResult, Message := 'Execution Result mismatch');
AssertEquals(Expected := ExpectedMotion, Actual := ActualMotion, Message := 'Motion Status mismatch');
AssertEquals(Expected := ExpectedWarnFault, Actual := ActualWarnFault, Message := 'Warning/Fault Flag mismatch');
AssertEquals(Expected := ExpectedDataField, Actual := ActualDataField, Message := 'Data Field mismatch');
AssertEquals(Expected := ExpectedChecksum, Actual := ActualChecksum, Message := 'Checksum mismatch');

TEST_FINISHED();
END_METHOD

METHOD PRIVATE GivenIdleReplyExpectCorrectFieldExtractionChecksum_1
VAR
    InputReply         : STRING := '@02 0 OK IDLE -- 0:8C';
    ExpectedAddress    : STRING := '02';
    ExpectedAxis       : STRING := '0';
    ExpectedResult     : STRING := 'OK';
    ExpectedMotion     : STRING := 'IDLE';
    ExpectedWarnFault  : STRING := '--';
    ExpectedDataField  : STRING := '0';
    ExpectedChecksum   : STRING := '8C';

    ActualAddress      : STRING;
    ActualAxis         : STRING;
    ActualResult       : STRING;
    ActualMotion       : STRING;
    ActualWarnFault    : STRING;
    ActualDataField    : STRING;
    ActualChecksum     : STRING;
END_VAR
TEST(__POUNAME());

// Execute field extraction
ActualAddress     := F_ExtractDeviceAddress(sInput := InputReply);
ActualAxis        := F_ExtractAxisNumber(sInput := InputReply);
ActualResult      := F_ZaberExtractExecutionResult(sInput := InputReply);
ActualMotion      := F_ExtractMotionStatus(sInput := InputReply);
ActualWarnFault   := F_ZaberExtractWarnFaultFlag(sInput := InputReply);
ActualDataField   := F_ExtractDataField(sInput := InputReply);
ActualChecksum    := F_ExtractMessageChecksum(sInput := InputReply);

// Assertions
AssertEquals(Expected := ExpectedAddress, Actual := ActualAddress, Message := 'Device Address mismatch');
AssertEquals(Expected := ExpectedAxis, Actual := ActualAxis, Message := 'Axis Number mismatch');
AssertEquals(Expected := ExpectedResult, Actual := ActualResult, Message := 'Execution Result mismatch');
AssertEquals(Expected := ExpectedMotion, Actual := ActualMotion, Message := 'Motion Status mismatch');
AssertEquals(Expected := ExpectedWarnFault, Actual := ActualWarnFault, Message := 'Warning/Fault Flag mismatch');
AssertEquals(Expected := ExpectedDataField, Actual := ActualDataField, Message := 'Data Field mismatch');
AssertEquals(Expected := ExpectedChecksum, Actual := ActualChecksum, Message := 'Checksum mismatch');

TEST_FINISHED();
END_METHOD

METHOD PRIVATE GivenIdleReplyExpectCorrectFieldExtractionNoChecksum
VAR
    InputReply         : STRING := '@02 0 OK IDLE -- 0 NA';
    ExpectedAddress    : STRING := '02';
    ExpectedAxis       : STRING := '0';
    ExpectedResult     : STRING := 'OK';
    ExpectedMotion     : STRING := 'IDLE';
    ExpectedWarnFault  : STRING := '--';
    ExpectedDataField  : STRING := '0 NA';
	ExpectedChecksum   : STRING := '';

    ActualAddress      : STRING;
    ActualAxis         : STRING;
    ActualResult       : STRING;
    ActualMotion       : STRING;
    ActualWarnFault    : STRING;
    ActualDataField    : STRING;
    ActualChecksum     : STRING;
END_VAR
TEST(__POUNAME());

// Execute field extraction
ActualAddress     := F_ExtractDeviceAddress(sInput := InputReply);
ActualAxis        := F_ExtractAxisNumber(sInput := InputReply);
ActualResult      := F_ZaberExtractExecutionResult(sInput := InputReply);
ActualMotion      := F_ExtractMotionStatus(sInput := InputReply);
ActualWarnFault   := F_ZaberExtractWarnFaultFlag(sInput := InputReply);
ActualDataField   := F_ExtractDataField(sInput := InputReply);
ActualChecksum    := F_ExtractMessageChecksum(sInput := InputReply);

// Assertions
AssertEquals(Expected := ExpectedAddress, Actual := ActualAddress, Message := 'Device Address mismatch');
AssertEquals(Expected := ExpectedAxis, Actual := ActualAxis, Message := 'Axis Number mismatch');
AssertEquals(Expected := ExpectedResult, Actual := ActualResult, Message := 'Execution Result mismatch');
AssertEquals(Expected := ExpectedMotion, Actual := ActualMotion, Message := 'Motion Status mismatch');
AssertEquals(Expected := ExpectedWarnFault, Actual := ActualWarnFault, Message := 'Warning/Fault Flag mismatch');
AssertEquals(Expected := ExpectedDataField, Actual := ActualDataField, Message := 'Data Field mismatch');
AssertEquals(Expected := ExpectedChecksum, Actual := ActualChecksum, Message := 'Checksum mismatch');

TEST_FINISHED();
END_METHOD

METHOD PRIVATE GivenNIReplyExpectCorrectFieldExtractionChecksum
VAR
    InputReply         : STRING := '@02 0 OK IDLE NI 0 NA:A0';
    ExpectedAddress    : STRING := '02';
    ExpectedAxis       : STRING := '0';
    ExpectedResult     : STRING := 'OK';
    ExpectedMotion     : STRING := 'IDLE';
    ExpectedWarnFault  : STRING := 'NI';
    ExpectedDataField  : STRING := '0 NA';
    ExpectedChecksum   : STRING := 'A0';

    ActualAddress      : STRING;
    ActualAxis         : STRING;
    ActualResult       : STRING;
    ActualMotion       : STRING;
    ActualWarnFault    : STRING;
    ActualDataField    : STRING;
    ActualChecksum     : STRING;
END_VAR
TEST(__POUNAME());

// Execute field extraction
ActualAddress     := F_ExtractDeviceAddress(sInput := InputReply);
ActualAxis        := F_ExtractAxisNumber(sInput := InputReply);
ActualResult      := F_ZaberExtractExecutionResult(sInput := InputReply);
ActualMotion      := F_ExtractMotionStatus(sInput := InputReply);
ActualWarnFault   := F_ZaberExtractWarnFaultFlag(sInput := InputReply);
ActualDataField   := F_ExtractDataField(sInput := InputReply);
ActualChecksum    := F_ExtractMessageChecksum(sInput := InputReply);

// Assertions
AssertEquals(Expected := ExpectedAddress, Actual := ActualAddress, Message := 'Device Address mismatch');
AssertEquals(Expected := ExpectedAxis, Actual := ActualAxis, Message := 'Axis Number mismatch');
AssertEquals(Expected := ExpectedResult, Actual := ActualResult, Message := 'Execution Result mismatch');
AssertEquals(Expected := ExpectedMotion, Actual := ActualMotion, Message := 'Motion Status mismatch');
AssertEquals(Expected := ExpectedWarnFault, Actual := ActualWarnFault, Message := 'Warning/Fault Flag mismatch');
AssertEquals(Expected := ExpectedDataField, Actual := ActualDataField, Message := 'Data Field mismatch');
AssertEquals(Expected := ExpectedChecksum, Actual := ActualChecksum, Message := 'Checksum mismatch');

TEST_FINISHED();
END_METHOD

METHOD PRIVATE GivenNIReplyExpectCorrectFieldExtractionNoChecksum
VAR
    InputReply         : STRING := '@02 0 OK IDLE NI 0 NA';
    ExpectedAddress    : STRING := '02';
    ExpectedAxis       : STRING := '0';
    ExpectedResult     : STRING := 'OK';
    ExpectedMotion     : STRING := 'IDLE';
    ExpectedWarnFault  : STRING := 'NI';
    ExpectedDataField  : STRING := '0 NA';
    ExpectedChecksum   : STRING := '';

    ActualAddress      : STRING;
    ActualAxis         : STRING;
    ActualResult       : STRING;
    ActualMotion       : STRING;
    ActualWarnFault    : STRING;
    ActualDataField    : STRING;
    ActualChecksum     : STRING;
END_VAR
TEST(__POUNAME());

// Execute field extraction
ActualAddress     := F_ExtractDeviceAddress(sInput := InputReply);
ActualAxis        := F_ExtractAxisNumber(sInput := InputReply);
ActualResult      := F_ZaberExtractExecutionResult(sInput := InputReply);
ActualMotion      := F_ExtractMotionStatus(sInput := InputReply);
ActualWarnFault   := F_ZaberExtractWarnFaultFlag(sInput := InputReply);
ActualDataField   := F_ExtractDataField(sInput := InputReply);
ActualChecksum    := F_ExtractMessageChecksum(sInput := InputReply);

// Assertions
AssertEquals(Expected := ExpectedAddress, Actual := ActualAddress, Message := 'Device Address mismatch');
AssertEquals(Expected := ExpectedAxis, Actual := ActualAxis, Message := 'Axis Number mismatch');
AssertEquals(Expected := ExpectedResult, Actual := ActualResult, Message := 'Execution Result mismatch');
AssertEquals(Expected := ExpectedMotion, Actual := ActualMotion, Message := 'Motion Status mismatch');
AssertEquals(Expected := ExpectedWarnFault, Actual := ActualWarnFault, Message := 'Warning/Fault Flag mismatch');
AssertEquals(Expected := ExpectedDataField, Actual := ActualDataField, Message := 'Data Field mismatch');
AssertEquals(Expected := ExpectedChecksum, Actual := ActualChecksum, Message := 'Checksum mismatch');

TEST_FINISHED();
END_METHOD

METHOD PRIVATE GivenReply_ExpectCorrectTokenization
VAR
    Input   : STRING := '@02 0 OK BUSY -- 0';
    Tokens  : ARRAY[1..16] OF STRING;
	i : INT;
	AccessibleToken1	: STRING := '@02';
	AccessibleToken2	: STRING := '0';
	AccessibleToken3	: STRING := 'OK';
	AccessibleToken4	: STRING := 'BUSY';
	AccessibleToken5	: STRING := '--';
	AccessibleToken6	: STRING := '0';
	AccessibleToken7	: STRING := '';
END_VAR
TEST(__POUNAME());

Tokens := F_ZaberSplitReplyTokensEx(sInput := Input);

// Assertions
AssertEquals(Expected := AccessibleToken1, Actual := Tokens[1], Message := 'Token 1 mismatch');
AssertEquals(Expected := AccessibleToken2, Actual := Tokens[2], Message := 'Token 2 mismatch');
AssertEquals(Expected := AccessibleToken3, Actual := Tokens[3], Message := 'Token 3 mismatch');
AssertEquals(Expected := AccessibleToken4, Actual := Tokens[4], Message := 'Token 4 mismatch');
AssertEquals(Expected := AccessibleToken5, Actual := Tokens[5], Message := 'Token 5 mismatch');
AssertEquals(Expected := AccessibleToken6, Actual := Tokens[6], Message := 'Token 6 mismatch');

// Check no extras
FOR i := 7 TO 16 DO
    AssertEquals(Expected := AccessibleToken7, Actual := Tokens[i], Message := CONCAT('Expected empty token at index ', DINT_TO_STRING(i)));
END_FOR

TEST_FINISHED();
END_METHOD

END_FUNCTION_BLOCK

// Zaber/Testing/FB_ZaberAxisTests
FUNCTION_BLOCK FB_ZaberAxisTests EXTENDS TcUnit.FB_TestSuite
VAR
END_VAR

END_FUNCTION_BLOCK

// Zaber/Testing/PRG_TEST
PROGRAM PRG_TEST
VAR
	StringHandlingTests	: FB_ValidateStringHandlingTests;
	ZaberAxisTests		: FB_ZaberAxisTests;
END_VAR

TcUnit.RUN();

END_PROGRAM

// MAIN
PROGRAM MAIN
VAR
	//ZaberGroup		: FB_ZaberSerialGroup;
	WebDrive		: FB_WebDrive;
END_VAR

//ZaberGroup.CyclicLogic();
WebDrive.CyclicLogic();

END_PROGRAM
